gfCNCPoint4[22804] = {X 353.6578, Y 29.0247, Z -6.3333, A 0.000, B 0.000, C 0.000 }
gfCNCPoint4[22805] = {X 353.9952, Y 27.8508, Z -6.3333, A 0.000, B 0.000, C 0.000 }
gfCNCPoint4[22806] = {X 354.2226, Y 26.4400, Z -6.3333, A 0.000, B 0.000, C 0.000 }
gfCNCPoint4[22807] = {X 354.3146, Y 25.0140, Z -6.3333, A 0.000, B 0.000, C 0.000 }
gfCNCPoint4[22808] = {X 354.2704, Y 23.5857, Z -6.3333, A 0.000, B 0.000, C 0.000 }
gfCNCPoint4[22809] = {X 354.0904, Y 22.1681, Z -6.3333, A 0.000, B 0.000, C 0.000 }
gfCNCPoint4[22810] = {X 353.8255, Y 21.0252, Z -6.3333, A 0.000, B 0.000, C 0.000 }
gfCNCPoint4[22811] = {X 353.4123, Y 19.9272, Z -6.3333, A 0.000, B 0.000, C 0.000 }
gfCNCPoint4[22812] = {X 352.8578, Y 18.8933, Z -6.3333, A 0.000, B 0.000, C 0.000 }
gfCNCPoint4[22813] = {X 352.1719, Y 17.9415, Z -6.3333, A 0.000, B 0.000, C 0.000 }
gfCNCPoint4[22814] = {X 351.4219, Y 17.1684, Z -6.3333, A 0.000, B 0.000, C 0.000 }
gfCNCPoint4[22815] = {X 350.5492, Y 16.5370, Z -6.3333, A 0.000, B 0.000, C 0.000 }
gfCNCPoint4[22816] = {X 349.5803, Y 16.0665, Z -6.3333, A 0.000, B 0.000, C 0.000 }
gfCNCPoint4[22817] = {X 348.5445, Y 15.7710, Z -6.3333, A 0.000, B 0.000, C 0.000 }
gfCNCPoint4[22818] = {X 347.1584, Y 15.5990, Z -6.3333, A 0.000, B 0.000, C 0.000 }
gfCNCPoint4[22819] = {X 345.7616, Y 15.6142, Z -6.3333, A 0.000, B 0.000, C 0.000 }
gfCNCPoint4[22820] = {X 344.3795, Y 15.8164, Z -6.3333, A 0.000, B 0.000, C 0.000 }
gfCNCPoint4[22821] = {X 343.0370, Y 16.2019, Z -6.3333, A 0.000, B 0.000, C 0.000 }
gfCNCPoint4[22822] = {X 341.7582, Y 16.7639, Z -6.3333, A 0.000, B 0.000, C 0.000 }
gfCNCPoint4[22823] = {X 341.3707, Y 18.0084, Z -6.3333, A 0.000, B 0.000, C 0.000 }
gfCNCPoint4[22824] = {X 340.7675, Y 19.1639, Z -6.3333, A 0.000, B 0.000, C 0.000 }
gfCNCPoint4[22825] = {X 339.9680, Y 20.1933, Z -6.3333, A 0.000, B 0.000, C 0.000 }
gfCNCPoint4[22826] = {X 338.9976, Y 21.0636, Z -6.3333, A 0.000, B 0.000, C 0.000 }
gfCNCPoint4[22827] = {X 338.2497, Y 21.6140, Z -6.3333, A 0.000, B 0.000, C 0.000 }
gfCNCPoint4[22828] = {X 337.8538, Y 21.8795, Z -6.3333, A 0.000, B 0.000, C 0.000 }
gfCNCPoint4[22829] = {X 337.4413, Y 22.1185, Z -6.3333, A 0.000, B 0.000, C 0.000 }
gfCNCPoint4[22830] = {X 336.3239, Y 22.6023, Z -6.3333, A 0.000, B 0.000, C 0.000 }
gfCNCPoint4[22831] = {X 335.1415, Y 22.8932, Z -6.3333, A 0.000, B 0.000, C 0.000 }
gfCNCPoint4[22832] = {X 333.9271, Y 22.9829, Z -6.3333, A 0.000, B 0.000, C 0.000 }
gfCNCPoint4[22833] = {X 332.7148, Y 22.8690, Z -6.3333, A 0.000, B 0.000, C 0.000 }
gfCNCPoint4[22834] = {X 331.5384, Y 22.5546, Z -6.3333, A 0.000, B 0.000, C 0.000 }
gfCNCPoint4[22835] = {X 330.4309, Y 22.0485, Z -6.3333, A 0.000, B 0.000, C 0.000 }
gfCNCPoint4[22836] = {X 329.5143, Y 21.4374, Z -6.3333, A 0.000, B 0.000, C 0.000 }
gfCNCPoint4[22837] = {X 328.7005, Y 20.6949, Z -6.3333, A 0.000, B 0.000, C 0.000 }
gfCNCPoint4[22838] = {X 328.0080, Y 19.8382, Z -6.3333, A 0.000, B 0.000, C 0.000 }
gfCNCPoint4[22839] = {X 327.4528, Y 18.8869, Z -6.3333, A 0.000, B 0.000, C 0.000 }
gfCNCPoint4[22840] = {X 323.9321, Y 11.6443, Z -6.3333, A 0.000, B 0.000, C 0.000 }
gfCNCPoint4[22841] = {X 323.5337, Y 10.6421, Z -6.3333, A 0.000, B 0.000, C 0.000 }
gfCNCPoint4[22842] = {X 323.2878, Y 9.5921, Z -6.3333, A 0.000, B 0.000, C 0.000 }
gfCNCPoint4[22843] = {X 323.1997, Y 8.5173, Z -6.3333, A 0.000, B 0.000, C 0.000 }
gfCNCPoint4[22844] = {X 323.2713, Y 7.4413, Z -6.3333, A 0.000, B 0.000, C 0.000 }
gfCNCPoint4[22845] = {X 323.4720, Y 6.4884, Z -6.3333, A 0.000, B 0.000, C 0.000 }
gfCNCPoint4[22846] = {X 323.7980, Y 5.5708, Z -6.3333, A 0.000, B 0.000, C 0.000 }
gfCNCPoint4[22847] = {X 324.2436, Y 4.7049, Z -6.3333, A 0.000, B 0.000, C 0.000 }
gfCNCPoint4[22848] = {X 168.0206, Y 4.7049, Z -6.3333, A 0.000, B 0.000, C 0.000 }
gfCNCPoint4[22849] = {X 168.0206, Y 9.5049, Z -6.3333, A 0.000, B 0.000, C 0.000 }
gfCNCPoint4[22850] = {X 166.5360, Y 9.5049, Z -6.3333, A 0.000, B 0.000, C 0.000 }
gfCNCPoint4[22851] = {X 166.5855, Y 9.9931, Z -6.3333, A 0.000, B 0.000, C 0.000 }
gfCNCPoint4[22852] = {X 166.6021, Y 10.4835, Z -6.3333, A 0.000, B 0.000, C 0.000 }
gfCNCPoint4[22853] = {X 166.6021, Y 13.0969, Z -6.3333, A 0.000, B 0.000, C 0.000 }
gfCNCPoint4[22854] = {X 166.8569, Y 11.8209, Z -6.3333, A 0.000, B 0.000, C 0.000 }
gfCNCPoint4[22855] = {X 167.3349, Y 10.6107, Z -6.3333, A 0.000, B 0.000, C 0.000 }
gfCNCPoint4[22856] = {X 168.0206, Y 9.5049, Z -6.3333, A 0.000, B 0.000, C 0.000 }
gfCNCPoint4[22857] = {X 168.0206, Y 7.1049, Z -6.3333, A 0.000, B 0.000, C 0.000 }
gfCNCPoint4[22858] = {X 162.8434, Y 7.1049, Z -6.3333, A 0.000, B 0.000, C 0.000 }
gfCNCPoint4[22859] = {X 163.4702, Y 7.9130, Z -6.3333, A 0.000, B 0.000, C 0.000 }
gfCNCPoint4[22860] = {X 163.9149, Y 8.8340, Z -6.3333, A 0.000, B 0.000, C 0.000 }
gfCNCPoint4[22861] = {X 164.1578, Y 9.8275, Z -6.3333, A 0.000, B 0.000, C 0.000 }
gfCNCPoint4[22862] = {X 164.1910, Y 10.1548, Z -6.3333, A 0.000, B 0.000, C 0.000 }
gfCNCPoint4[22863] = {X 164.2021, Y 10.4835, Z -6.3333, A 0.000, B 0.000, C 0.000 }
gfCNCPoint4[22864] = {X 164.2021, Y 17.4615, Z -6.3333, A 0.000, B 0.000, C 0.000 }
gfCNCPoint4[22865] = {X 164.1140, Y 18.3847, Z -6.3333, A 0.000, B 0.000, C 0.000 }
gfCNCPoint4[22866] = {X 163.8528, Y 19.2745, Z -6.3333, A 0.000, B 0.000, C 0.000 }
gfCNCPoint4[22867] = {X 163.4280, Y 20.0989, Z -6.3333, A 0.000, B 0.000, C 0.000 }
gfCNCPoint4[22868] = {X 162.8550, Y 20.8280, Z -6.3333, A 0.000, B 0.000, C 0.000 }
gfCNCPoint4[22869] = {X 162.1544, Y 21.4355, Z -6.3333, A 0.000, B 0.000, C 0.000 }
gfCNCPoint4[22870] = {X 161.3515, Y 21.8996, Z -6.3333, A 0.000, B 0.000, C 0.000 }
gfCNCPoint4[22871] = {X 160.4753, Y 22.2033, Z -6.3333, A 0.000, B 0.000, C 0.000 }
gfCNCPoint4[22872] = {X 162.1767, Y 29.1994, Z -6.3333, A 0.000, B 0.000, C 0.000 }
gfCNCPoint4[22873] = {X 161.1138, Y 29.4079, Z -6.3333, A 0.000, B 0.000, C 0.000 }
gfCNCPoint4[22874] = {X 160.0364, Y 29.5204, Z -6.3333, A 0.000, B 0.000, C 0.000 }
gfCNCPoint4[22875] = {X 160.0359, Y 38.3363, Z -6.3333, A 0.000, B 0.000, C 0.000 }
gfCNCPoint4[22876] = {X 160.6841, Y 39.6935, Z -6.3333, A 0.000, B 0.000, C 0.000 }
gfCNCPoint4[22877] = {X 161.1590, Y 41.1206, Z -6.3333, A 0.000, B 0.000, C 0.000 }
gfCNCPoint4[22878] = {X 162.0525, Y 41.1205, Z -6.3333, A 0.000, B 0.000, C 0.000 }
gfCNCPoint4[22879] = {X 161.8701, Y 40.3466, Z -6.3333, A 0.000, B 0.000, C 0.000 }
gfCNCPoint4[22880] = {X 161.7176, Y 39.5664, Z -6.3333, A 0.000, B 0.000, C 0.000 }
gfCNCPoint4[22881] = {X 161.5943, Y 38.7924, Z -6.3333, A 0.000, B 0.000, C 0.000 }
gfCNCPoint4[22882] = {X 161.3800, Y 36.8680, Z -6.3333, A 0.000, B 0.000, C 0.000 }
gfCNCPoint4[22883] = {X 161.3313, Y 34.9322, Z -6.3333, A 0.000, B 0.000, C 0.000 }
gfCNCPoint4[22884] = {X 161.4486, Y 32.9994, Z -6.3333, A 0.000, B 0.000, C 0.000 }
gfCNCPoint4[22885] = {X 161.7311, Y 31.0838, Z -6.3333, A 0.000, B 0.000, C 0.000 }
gfCNCPoint4[22886] = {X 162.1767, Y 29.1994, Z -6.3333, A 0.000, B 0.000, C 0.000 }
gfCNCPoint4[22887] = {X 161.6096, Y 26.8674, Z -6.3333, A 0.000, B 0.000, C 0.000 }
gfCNCPoint4[22888] = {X 160.4740, Y 27.0728, Z -6.3333, A 0.000, B 0.000, C 0.000 }
gfCNCPoint4[22889] = {X 159.3220, Y 27.1415, Z -6.3333, A 0.000, B 0.000, C 0.000 }
gfCNCPoint4[22890] = {X 158.6595, Y 27.1415, Z -6.3333, A 0.000, B 0.000, C 0.000 }
gfCNCPoint4[22891] = {X 158.1473, Y 27.1261, Z -6.3333, A 0.000, B 0.000, C 0.000 }
gfCNCPoint4[22892] = {X 157.6365, Y 27.0837, Z -6.3333, A 0.000, B 0.000, C 0.000 }
gfCNCPoint4[22893] = {X 157.6359, Y 38.9959, Z -6.3333, A 0.000, B 0.000, C 0.000 }
gfCNCPoint4[22894] = {X 158.2197, Y 40.0483, Z -6.3333, A 0.000, B 0.000, C 0.000 }
gfCNCPoint4[22895] = {X 158.6689, Y 41.1648, Z -6.3333, A 0.000, B 0.000, C 0.000 }
gfCNCPoint4[22896] = {X 158.9765, Y 42.3283, Z -6.3333, A 0.000, B 0.000, C 0.000 }
gfCNCPoint4[22897] = {X 159.1377, Y 43.5209, Z -6.3333, A 0.000, B 0.000, C 0.000 }
gfCNCPoint4[22898] = {X 165.4263, Y 43.5200, Z -6.3333, A 0.000, B 0.000, C 0.000 }
gfCNCPoint4[22899] = {X 164.8372, Y 42.0454, Z -6.3333, A 0.000, B 0.000, C 0.000 }
gfCNCPoint4[22900] = {X 164.3775, Y 40.5256, Z -6.3333, A 0.000, B 0.000, C 0.000 }
gfCNCPoint4[22901] = {X 164.2182, Y 39.8499, Z -6.3333, A 0.000, B 0.000, C 0.000 }
gfCNCPoint4[22902] = {X 164.0845, Y 39.1688, Z -6.3333, A 0.000, B 0.000, C 0.000 }
gfCNCPoint4[22903] = {X 163.9653, Y 38.4202, Z -6.3333, A 0.000, B 0.000, C 0.000 }
gfCNCPoint4[22904] = {X 163.7495, Y 36.2693, Z -6.3333, A 0.000, B 0.000, C 0.000 }
gfCNCPoint4[22905] = {X 163.7649, Y 34.1077, Z -6.3333, A 0.000, B 0.000, C 0.000 }
gfCNCPoint4[22906] = {X 164.0116, Y 31.9602, Z -6.3333, A 0.000, B 0.000, C 0.000 }
gfCNCPoint4[22907] = {X 164.4865, Y 29.8513, Z -6.3333, A 0.000, B 0.000, C 0.000 }
gfCNCPoint4[22908] = {X 164.8367, Y 28.7352, Z -6.3333, A 0.000, B 0.000, C 0.000 }
gfCNCPoint4[22909] = {X 165.2511, Y 27.6412, Z -6.3333, A 0.000, B 0.000, C 0.000 }
gfCNCPoint4[22910] = {X 165.8680, Y 26.3084, Z -6.3333, A 0.000, B 0.000, C 0.000 }
gfCNCPoint4[22911] = {X 166.6029, Y 25.0369, Z -6.3333, A 0.000, B 0.000, C 0.000 }
gfCNCPoint4[22912] = {X 167.4499, Y 23.8371, Z -6.3333, A 0.000, B 0.000, C 0.000 }
gfCNCPoint4[22913] = {X 167.1640, Y 23.1367, Z -6.3333, A 0.000, B 0.000, C 0.000 }
gfCNCPoint4[22914] = {X 166.2875, Y 24.1835, Z -6.3333, A 0.000, B 0.000, C 0.000 }
gfCNCPoint4[22915] = {X 165.2726, Y 25.0966, Z -6.3333, A 0.000, B 0.000, C 0.000 }
gfCNCPoint4[22916] = {X 164.1393, Y 25.8578, Z -6.3333, A 0.000, B 0.000, C 0.000 }
gfCNCPoint4[22917] = {X 162.9101, Y 26.4520, Z -6.3333, A 0.000, B 0.000, C 0.000 }
gfCNCPoint4[22918] = {X 161.6096, Y 26.8674, Z -6.3333, A 0.000, B 0.000, C 0.000 }
gfCNCPoint4[22919] = {X 161.0424, Y 24.5353, Z -6.3333, A 0.000, B 0.000, C 0.000 }
gfCNCPoint4[22920] = {X 160.1884, Y 24.6898, Z -6.3333, A 0.000, B 0.000, C 0.000 }
gfCNCPoint4[22921] = {X 159.3220, Y 24.7415, Z -6.3333, A 0.000, B 0.000, C 0.000 }
gfCNCPoint4[22922] = {X 158.6684, Y 24.7415, Z -6.3333, A 0.000, B 0.000, C 0.000 }
gfCNCPoint4[22923] = {X 158.2827, Y 24.7299, Z -6.3333, A 0.000, B 0.000, C 0.000 }
gfCNCPoint4[22924] = {X 157.8982, Y 24.6980, Z -6.3333, A 0.000, B 0.000, C 0.000 }
gfCNCPoint4[22925] = {X 156.9782, Y 24.5371, Z -6.3333, A 0.000, B 0.000, C 0.000 }
gfCNCPoint4[22926] = {X 156.0862, Y 24.2602, Z -6.3333, A 0.000, B 0.000, C 0.000 }
gfCNCPoint4[22927] = {X 155.2367, Y 23.8718, Z -6.3333, A 0.000, B 0.000, C 0.000 }
gfCNCPoint4[22928] = {X 155.2358, Y 39.7518, Z -6.3333, A 0.000, B 0.000, C 0.000 }
gfCNCPoint4[22929] = {X 155.8266, Y 40.6435, Z -6.3333, A 0.000, B 0.000, C 0.000 }
gfCNCPoint4[22930] = {X 156.2808, Y 41.6118, Z -6.3333, A 0.000, B 0.000, C 0.000 }
gfCNCPoint4[22931] = {X 156.5888, Y 42.6361, Z -6.3333, A 0.000, B 0.000, C 0.000 }
gfCNCPoint4[22932] = {X 156.7440, Y 43.6944, Z -6.3333, A 0.000, B 0.000, C 0.000 }
gfCNCPoint4[22933] = {X 156.7580, Y 43.9481, Z -6.3333, A 0.000, B 0.000, C 0.000 }
gfCNCPoint4[22934] = {X 156.7631, Y 44.2022, Z -6.3333, A 0.000, B 0.000, C 0.000 }
gfCNCPoint4[22935] = {X 156.7629, Y 45.0588, Z -6.3333, A 0.000, B 0.000, C 0.000 }
gfCNCPoint4[22936] = {X 156.7352, Y 45.6370, Z -6.3333, A 0.000, B 0.000, C 0.000 }
gfCNCPoint4[22937] = {X 156.6616, Y 46.2112, Z -6.3333, A 0.000, B 0.000, C 0.000 }
gfCNCPoint4[22938] = {X 157.9054, Y 46.0005, Z -6.3333, A 0.000, B 0.000, C 0.000 }
gfCNCPoint4[22939] = {X 159.1643, Y 45.9207, Z -6.3333, A 0.000, B 0.000, C 0.000 }
gfCNCPoint4[22940] = {X 159.2311, Y 45.9202, Z -6.3333, A 0.000, B 0.000, C 0.000 }
gfCNCPoint4[22941] = {X 159.2980, Y 45.9200, Z -6.3333, A 0.000, B 0.000, C 0.000 }
gfCNCPoint4[22942] = {X 169.6793, Y 45.9200, Z -6.3333, A 0.000, B 0.000, C 0.000 }
gfCNCPoint4[22943] = {X 168.8981, Y 44.8498, Z -6.3333, A 0.000, B 0.000, C 0.000 }
gfCNCPoint4[22944] = {X 168.2083, Y 43.7186, Z -6.3333, A 0.000, B 0.000, C 0.000 }
gfCNCPoint4[22945] = {X 167.6145, Y 42.5342, Z -6.3333, A 0.000, B 0.000, C 0.000 }
gfCNCPoint4[22946] = {X 167.1237, Y 41.3128, Z -6.3333, A 0.000, B 0.000, C 0.000 }
gfCNCPoint4[22947] = {X 166.7350, Y 40.0551, Z -6.3333, A 0.000, B 0.000, C 0.000 }
gfCNCPoint4[22948] = {X 166.4512, Y 38.7697, Z -6.3333, A 0.000, B 0.000, C 0.000 }
gfCNCPoint4[22949] = {X 166.3363, Y 38.0482, Z -6.3333, A 0.000, B 0.000, C 0.000 }
gfCNCPoint4[22950] = {X 166.1452, Y 36.1222, Z -6.3333, A 0.000, B 0.000, C 0.000 }
gfCNCPoint4[22951] = {X 166.1647, Y 34.1868, Z -6.3333, A 0.000, B 0.000, C 0.000 }
gfCNCPoint4[22952] = {X 166.3944, Y 32.2650, Z -6.3333, A 0.000, B 0.000, C 0.000 }
gfCNCPoint4[22953] = {X 166.8316, Y 30.3795, Z -6.3333, A 0.000, B 0.000, C 0.000 }
gfCNCPoint4[22954] = {X 167.4712, Y 28.5528, Z -6.3333, A 0.000, B 0.000, C 0.000 }
gfCNCPoint4[22955] = {X 168.2320, Y 26.9825, Z -6.3333, A 0.000, B 0.000, C 0.000 }
gfCNCPoint4[22956] = {X 169.1846, Y 25.5206, Z -6.3333, A 0.000, B 0.000, C 0.000 }
gfCNCPoint4[22957] = {X 170.3139, Y 24.1904, Z -6.3333, A 0.000, B 0.000, C 0.000 }
gfCNCPoint4[22958] = {X 169.9864, Y 23.6220, Z -6.3333, A 0.000, B 0.000, C 0.000 }
gfCNCPoint4[22959] = {X 169.7113, Y 23.0264, Z -6.3333, A 0.000, B 0.000, C 0.000 }
gfCNCPoint4[22960] = {X 167.1001, Y 16.6309, Z -6.3333, A 0.000, B 0.000, C 0.000 }
gfCNCPoint4[22961] = {X 166.7820, Y 15.6636, Z -6.3333, A 0.000, B 0.000, C 0.000 }
gfCNCPoint4[22962] = {X 166.6021, Y 14.6613, Z -6.3333, A 0.000, B 0.000, C 0.000 }
gfCNCPoint4[22963] = {X 166.6021, Y 17.4615, Z -6.3333, A 0.000, B 0.000, C 0.000 }
gfCNCPoint4[22964] = {X 166.5130, Y 18.5970, Z -6.3333, A 0.000, B 0.000, C 0.000 }
gfCNCPoint4[22965] = {X 166.2479, Y 19.7047, Z -6.3333, A 0.000, B 0.000, C 0.000 }
gfCNCPoint4[22966] = {X 165.8132, Y 20.7575, Z -6.3333, A 0.000, B 0.000, C 0.000 }
gfCNCPoint4[22967] = {X 165.2197, Y 21.7296, Z -6.3333, A 0.000, B 0.000, C 0.000 }
gfCNCPoint4[22968] = {X 164.3790, Y 22.6986, Z -6.3333, A 0.000, B 0.000, C 0.000 }
gfCNCPoint4[22969] = {X 163.3812, Y 23.5049, Z -6.3333, A 0.000, B 0.000, C 0.000 }
gfCNCPoint4[22970] = {X 162.2574, Y 24.1236, Z -6.3333, A 0.000, B 0.000, C 0.000 }
gfCNCPoint4[22971] = {X 161.0424, Y 24.5353, Z -6.3333, A 0.000, B 0.000, C 0.000 }
gfCNCPoint4[22972] = {X 160.4753, Y 22.2033, Z -6.3333, A 0.000, B 0.000, C 0.000 }
gfCNCPoint4[22973] = {X 159.9028, Y 22.3069, Z -6.3333, A 0.000, B 0.000, C 0.000 }
gfCNCPoint4[22974] = {X 159.3220, Y 22.3415, Z -6.3333, A 0.000, B 0.000, C 0.000 }
gfCNCPoint4[22975] = {X 158.6772, Y 22.3415, Z -6.3333, A 0.000, B 0.000, C 0.000 }
gfCNCPoint4[22976] = {X 157.8803, Y 22.2735, Z -6.3333, A 0.000, B 0.000, C 0.000 }
gfCNCPoint4[22977] = {X 157.1051, Y 22.0770, Z -6.3333, A 0.000, B 0.000, C 0.000 }
gfCNCPoint4[22978] = {X 156.3720, Y 21.7573, Z -6.3333, A 0.000, B 0.000, C 0.000 }
gfCNCPoint4[22979] = {X 155.5228, Y 21.1795, Z -6.3333, A 0.000, B 0.000, C 0.000 }
gfCNCPoint4[22980] = {X 154.8124, Y 20.4377, Z -6.3333, A 0.000, B 0.000, C 0.000 }
gfCNCPoint4[22981] = {X 152.8369, Y 20.4384, Z -6.3333, A 0.000, B 0.000, C 0.000 }
gfCNCPoint4[22982] = {X 152.8358, Y 40.6543, Z -6.3333, A 0.000, B 0.000, C 0.000 }
gfCNCPoint4[22983] = {X 153.1748, Y 41.0209, Z -6.3333, A 0.000, B 0.000, C 0.000 }
gfCNCPoint4[22984] = {X 153.6800, Y 41.7251, Z -6.3333, A 0.000, B 0.000, C 0.000 }
gfCNCPoint4[22985] = {X 154.0535, Y 42.5072, Z -6.3333, A 0.000, B 0.000, C 0.000 }
gfCNCPoint4[22986] = {X 154.2836, Y 43.3429, Z -6.3333, A 0.000, B 0.000, C 0.000 }
gfCNCPoint4[22987] = {X 154.3631, Y 44.2060, Z -6.3333, A 0.000, B 0.000, C 0.000 }
gfCNCPoint4[22988] = {X 154.3629, Y 45.0469, Z -6.3333, A 0.000, B 0.000, C 0.000 }
gfCNCPoint4[22989] = {X 154.3440, Y 45.4308, Z -6.3333, A 0.000, B 0.000, C 0.000 }
gfCNCPoint4[22990] = {X 154.2951, Y 45.8119, Z -6.3333, A 0.000, B 0.000, C 0.000 }
gfCNCPoint4[22991] = {X 154.0370, Y 46.7541, Z -6.3333, A 0.000, B 0.000, C 0.000 }
gfCNCPoint4[22992] = {X 153.5963, Y 47.6260, Z -6.3333, A 0.000, B 0.000, C 0.000 }
gfCNCPoint4[22993] = {X 152.9909, Y 48.3926, Z -6.3333, A 0.000, B 0.000, C 0.000 }
gfCNCPoint4[22994] = {X 152.2448, Y 49.0233, Z -6.3333, A 0.000, B 0.000, C 0.000 }
gfCNCPoint4[22995] = {X 151.3881, Y 49.4928, Z -6.3333, A 0.000, B 0.000, C 0.000 }
gfCNCPoint4[22996] = {X 150.4551, Y 49.7822, Z -6.3333, A 0.000, B 0.000, C 0.000 }
gfCNCPoint4[22997] = {X 149.4831, Y 49.8800, Z -6.3333, A 0.000, B 0.000, C 0.000 }
gfCNCPoint4[22998] = {X 143.0396, Y 49.8800, Z -6.3333, A 0.000, B 0.000, C 0.000 }
gfCNCPoint4[22999] = {X 142.0923, Y 49.7872, Z -6.3333, A 0.000, B 0.000, C 0.000 }
gfCNCPoint4[23000] = {X 141.1811, Y 49.5122, Z -6.3333, A 0.000, B 0.000, C 0.000 }
gfCNCPoint4[23001] = {X 140.3405, Y 49.0656, Z -6.3333, A 0.000, B 0.000, C 0.000 }
gfCNCPoint4[23002] = {X 139.6026, Y 48.4643, Z -6.3333, A 0.000, B 0.000, C 0.000 }
gfCNCPoint4[23003] = {X 138.9955, Y 47.7312, Z -6.3333, A 0.000, B 0.000, C 0.000 }
gfCNCPoint4[23004] = {X 138.5423, Y 46.8942, Z -6.3333, A 0.000, B 0.000, C 0.000 }
gfCNCPoint4[23005] = {X 138.2601, Y 45.9852, Z -6.3333, A 0.000, B 0.000, C 0.000 }
gfCNCPoint4[23006] = {X 138.1598, Y 45.0386, Z -6.3333, A 0.000, B 0.000, C 0.000 }
gfCNCPoint4[23007] = {X 138.1601, Y 44.1416, Z -6.3333, A 0.000, B 0.000, C 0.000 }
gfCNCPoint4[23008] = {X 138.2148, Y 43.4769, Z -6.3333, A 0.000, B 0.000, C 0.000 }
gfCNCPoint4[23009] = {X 138.3597, Y 42.8258, Z -6.3333, A 0.000, B 0.000, C 0.000 }
gfCNCPoint4[23010] = {X 129.1532, Y 40.1052, Z -6.3333, A 0.000, B 0.000, C 0.000 }
gfCNCPoint4[23011] = {X 129.5665, Y 38.9035, Z -6.3333, A 0.000, B 0.000, C 0.000 }
gfCNCPoint4[23012] = {X 130.0836, Y 37.7426, Z -6.3333, A 0.000, B 0.000, C 0.000 }
gfCNCPoint4[23013] = {X 130.0836, Y 31.6021, Z -6.3333, A 0.000, B 0.000, C 0.000 }
gfCNCPoint4[23014] = {X 129.2064, Y 31.3798, Z -6.3333, A 0.000, B 0.000, C 0.000 }
gfCNCPoint4[23015] = {X 128.3449, Y 31.1031, Z -6.3333, A 0.000, B 0.000, C 0.000 }
gfCNCPoint4[23016] = {X 128.3447, Y 38.3302, Z -6.3333, A 0.000, B 0.000, C 0.000 }
gfCNCPoint4[23017] = {X 128.7849, Y 39.2014, Z -6.3333, A 0.000, B 0.000, C 0.000 }
gfCNCPoint4[23018] = {X 129.1532, Y 40.1052, Z -6.3333, A 0.000, B 0.000, C 0.000 }
gfCNCPoint4[23019] = {X 131.4548, Y 40.7854, Z -6.3333, A 0.000, B 0.000, C 0.000 }
gfCNCPoint4[23020] = {X 131.9017, Y 39.5320, Z -6.3333, A 0.000, B 0.000, C 0.000 }
gfCNCPoint4[23021] = {X 132.4836, Y 38.3354, Z -6.3333, A 0.000, B 0.000, C 0.000 }
gfCNCPoint4[23022] = {X 132.4836, Y 29.5202, Z -6.3333, A 0.000, B 0.000, C 0.000 }
gfCNCPoint4[23023] = {X 131.3526, Y 29.3993, Z -6.3333, A 0.000, B 0.000, C 0.000 }
gfCNCPoint4[23024] = {X 130.2380, Y 29.1726, Z -6.3333, A 0.000, B 0.000, C 0.000 }
gfCNCPoint4[23025] = {X 129.1497, Y 28.8421, Z -6.3333, A 0.000, B 0.000, C 0.000 }
gfCNCPoint4[23026] = {X 128.0253, Y 28.3768, Z -6.3333, A 0.000, B 0.000, C 0.000 }
gfCNCPoint4[23027] = {X 126.9534, Y 27.8007, Z -6.3333, A 0.000, B 0.000, C 0.000 }
gfCNCPoint4[23028] = {X 125.9449, Y 27.1197, Z -6.3333, A 0.000, B 0.000, C 0.000 }
gfCNCPoint4[23029] = {X 125.9447, Y 38.9907, Z -6.3333, A 0.000, B 0.000, C 0.000 }
gfCNCPoint4[23030] = {X 126.4741, Y 39.9291, Z -6.3333, A 0.000, B 0.000, C 0.000 }
gfCNCPoint4[23031] = {X 126.8960, Y 40.9205, Z -6.3333, A 0.000, B 0.000, C 0.000 }
gfCNCPoint4[23032] = {X 127.2098, Y 41.9730, Z -6.3333, A 0.000, B 0.000, C 0.000 }
gfCNCPoint4[23033] = {X 127.4025, Y 43.0542, Z -6.3333, A 0.000, B 0.000, C 0.000 }
gfCNCPoint4[23034] = {X 127.4714, Y 44.1502, Z -6.3333, A 0.000, B 0.000, C 0.000 }
gfCNCPoint4[23035] = {X 127.4716, Y 45.0000, Z -6.3333, A 0.000, B 0.000, C 0.000 }
gfCNCPoint4[23036] = {X 127.4070, Y 46.1159, Z -6.3333, A 0.000, B 0.000, C 0.000 }
gfCNCPoint4[23037] = {X 127.2143, Y 47.2168, Z -6.3333, A 0.000, B 0.000, C 0.000 }
gfCNCPoint4[23038] = {X 126.8960, Y 48.2883, Z -6.3333, A 0.000, B 0.000, C 0.000 }
gfCNCPoint4[23039] = {X 126.2883, Y 49.6376, Z -6.3333, A 0.000, B 0.000, C 0.000 }
gfCNCPoint4[23040] = {X 125.4821, Y 50.8786, Z -6.3333, A 0.000, B 0.000, C 0.000 }
gfCNCPoint4[23041] = {X 124.4962, Y 51.9821, Z -6.3333, A 0.000, B 0.000, C 0.000 }
gfCNCPoint4[23042] = {X 123.3536, Y 52.9225, Z -6.3333, A 0.000, B 0.000, C 0.000 }
gfCNCPoint4[23043] = {X 122.0810, Y 53.6778, Z -6.3333, A 0.000, B 0.000, C 0.000 }
gfCNCPoint4[23044] = {X 120.7081, Y 54.2302, Z -6.3333, A 0.000, B 0.000, C 0.000 }
gfCNCPoint4[23045] = {X 119.2671, Y 54.5669, Z -6.3333, A 0.000, B 0.000, C 0.000 }
gfCNCPoint4[23046] = {X 117.7916, Y 54.6800, Z -6.3333, A 0.000, B 0.000, C 0.000 }
gfCNCPoint4[23047] = {X 111.9185, Y 54.6800, Z -6.3333, A 0.000, B 0.000, C 0.000 }
gfCNCPoint4[23048] = {X 111.7456, Y 54.6785, Z -6.3333, A 0.000, B 0.000, C 0.000 }
gfCNCPoint4[23049] = {X 111.5728, Y 54.6738, Z -6.3333, A 0.000, B 0.000, C 0.000 }
gfCNCPoint4[23050] = {X 111.0585, Y 69.0646, Z -6.3333, A 0.000, B 0.000, C 0.000 }
gfCNCPoint4[23051] = {X 109.0296, Y 68.9061, Z -6.3333, A 0.000, B 0.000, C 0.000 }
gfCNCPoint4[23052] = {X 107.0213, Y 68.5768, Z -6.3333, A 0.000, B 0.000, C 0.000 }
gfCNCPoint4[23053] = {X 105.0765, Y 68.8983, Z -6.3333, A 0.000, B 0.000, C 0.000 }
gfCNCPoint4[23054] = {X 103.1119, Y 69.0597, Z -6.3333, A 0.000, B 0.000, C 0.000 }
gfCNCPoint4[23055] = {X 101.1407, Y 69.0599, Z -6.3333, A 0.000, B 0.000, C 0.000 }
gfCNCPoint4[23056] = {X 99.1761, Y 68.8989, Z -6.3333, A 0.000, B 0.000, C 0.000 }
gfCNCPoint4[23057] = {X 97.2313, Y 68.5777, Z -6.3333, A 0.000, B 0.000, C 0.000 }
gfCNCPoint4[23058] = {X 95.6131, Y 68.8563, Z -6.3333, A 0.000, B 0.000, C 0.000 }
gfCNCPoint4[23059] = {X 93.9796, Y 69.0240, Z -6.3333, A 0.000, B 0.000, C 0.000 }
gfCNCPoint4[23060] = {X 92.3385, Y 69.0800, Z -6.3333, A 0.000, B 0.000, C 0.000 }
gfCNCPoint4[23061] = {X 86.6884, Y 69.0800, Z -6.3333, A 0.000, B 0.000, C 0.000 }
gfCNCPoint4[23062] = {X 84.7316, Y 70.2669, Z -6.3333, A 0.000, B 0.000, C 0.000 }
gfCNCPoint4[23063] = {X 82.6869, Y 71.2951, Z -6.3333, A 0.000, B 0.000, C 0.000 }
gfCNCPoint4[23064] = {X 107.2714, Y 71.2951, Z -6.3333, A 0.000, B 0.000, C 0.000 }
gfCNCPoint4[23065] = {X 109.1257, Y 70.1133, Z -6.3333, A 0.000, B 0.000, C 0.000 }
gfCNCPoint4[23066] = {X 111.0585, Y 69.0646, Z -6.3333, A 0.000, B 0.000, C 0.000 }
gfCNCPoint4[23067] = {X 111.1442, Y 66.6662, Z -6.3333, A 0.000, B 0.000, C 0.000 }
gfCNCPoint4[23068] = {X 109.0696, Y 66.4920, Z -6.3333, A 0.000, B 0.000, C 0.000 }
gfCNCPoint4[23069] = {X 107.0213, Y 66.1197, Z -6.3333, A 0.000, B 0.000, C 0.000 }
gfCNCPoint4[23070] = {X 105.0796, Y 66.4776, Z -6.3333, A 0.000, B 0.000, C 0.000 }
gfCNCPoint4[23071] = {X 103.1135, Y 66.6574, Z -6.3333, A 0.000, B 0.000, C 0.000 }
gfCNCPoint4[23072] = {X 101.1392, Y 66.6576, Z -6.3333, A 0.000, B 0.000, C 0.000 }
gfCNCPoint4[23073] = {X 99.1730, Y 66.4782, Z -6.3333, A 0.000, B 0.000, C 0.000 }
gfCNCPoint4[23074] = {X 97.2313, Y 66.1207, Z -6.3333, A 0.000, B 0.000, C 0.000 }
gfCNCPoint4[23075] = {X 95.6161, Y 66.4308, Z -6.3333, A 0.000, B 0.000, C 0.000 }
gfCNCPoint4[23076] = {X 93.9821, Y 66.6176, Z -6.3333, A 0.000, B 0.000, C 0.000 }
gfCNCPoint4[23077] = {X 92.3385, Y 66.6800, Z -6.3333, A 0.000, B 0.000, C 0.000 }
gfCNCPoint4[23078] = {X 85.9487, Y 66.6800, Z -6.3333, A 0.000, B 0.000, C 0.000 }
gfCNCPoint4[23079] = {X 83.8779, Y 67.9936, Z -6.3333, A 0.000, B 0.000, C 0.000 }
gfCNCPoint4[23080] = {X 81.6945, Y 69.1099, Z -6.3333, A 0.000, B 0.000, C 0.000 }
gfCNCPoint4[23081] = {X 79.6015, Y 69.9548, Z -6.3333, A 0.000, B 0.000, C 0.000 }
gfCNCPoint4[23082] = {X 77.4442, Y 70.6184, Z -6.3333, A 0.000, B 0.000, C 0.000 }
gfCNCPoint4[23083] = {X 75.2382, Y 71.0959, Z -6.3333, A 0.000, B 0.000, C 0.000 }
gfCNCPoint4[23084] = {X 72.9995, Y 71.3838, Z -6.3333, A 0.000, B 0.000, C 0.000 }
gfCNCPoint4[23085] = {X 70.7445, Y 71.4800, Z -6.3333, A 0.000, B 0.000, C 0.000 }
gfCNCPoint4[23086] = {X 64.1851, Y 71.4800, Z -6.3333, A 0.000, B 0.000, C 0.000 }
gfCNCPoint4[23087] = {X 62.0752, Y 71.3958, Z -6.3333, A 0.000, B 0.000, C 0.000 }
gfCNCPoint4[23088] = {X 59.9787, Y 71.1438, Z -6.3333, A 0.000, B 0.000, C 0.000 }
gfCNCPoint4[23089] = {X 57.9089, Y 70.7255, Z -6.3333, A 0.000, B 0.000, C 0.000 }
gfCNCPoint4[23090] = {X 55.8790, Y 70.1436, Z -6.3333, A 0.000, B 0.000, C 0.000 }
gfCNCPoint4[23091] = {X 53.8492, Y 70.7255, Z -6.3333, A 0.000, B 0.000, C 0.000 }
gfCNCPoint4[23092] = {X 51.7794, Y 71.1438, Z -6.3333, A 0.000, B 0.000, C 0.000 }
gfCNCPoint4[23093] = {X 49.6829, Y 71.3958, Z -6.3333, A 0.000, B 0.000, C 0.000 }
gfCNCPoint4[23094] = {X 47.5729, Y 71.4800, Z -6.3333, A 0.000, B 0.000, C 0.000 }
gfCNCPoint4[23095] = {X 40.6393, Y 71.4800, Z -6.3333, A 0.000, B 0.000, C 0.000 }
gfCNCPoint4[23096] = {X 38.8056, Y 71.4164, Z -6.3333, A 0.000, B 0.000, C 0.000 }
gfCNCPoint4[23097] = {X 36.9807, Y 71.2260, Z -6.3333, A 0.000, B 0.000, C 0.000 }
gfCNCPoint4[23098] = {X 34.3981, Y 72.0359, Z -6.3333, A 0.000, B 0.000, C 0.000 }
gfCNCPoint4[23099] = {X 31.7544, Y 72.6161, Z -6.3333, A 0.000, B 0.000, C 0.000 }
gfCNCPoint4[23100] = {X 30.3306, Y 73.1752, Z -6.3333, A 0.000, B 0.000, C 0.000 }
gfCNCPoint4[23101] = {X 28.8922, Y 73.6951, Z -6.3333, A 0.000, B 0.000, C 0.000 }
gfCNCPoint4[23102] = {X 108.0336, Y 73.6951, Z -6.3333, A 0.000, B 0.000, C 0.000 }
gfCNCPoint4[23103] = {X 110.0294, Y 72.3691, Z -6.3333, A 0.000, B 0.000, C 0.000 }
gfCNCPoint4[23104] = {X 112.1282, Y 71.2131, Z -6.3333, A 0.000, B 0.000, C 0.000 }
gfCNCPoint4[23105] = {X 113.1260, Y 70.7398, Z -6.3333, A 0.000, B 0.000, C 0.000 }
gfCNCPoint4[23106] = {X 114.1413, Y 70.3051, Z -6.3333, A 0.000, B 0.000, C 0.000 }
gfCNCPoint4[23107] = {X 117.4424, Y 66.6800, Z -6.3333, A 0.000, B 0.000, C 0.000 }
gfCNCPoint4[23108] = {X 111.9185, Y 66.6800, Z -6.3333, A 0.000, B 0.000, C 0.000 }
gfCNCPoint4[23109] = {X 111.5313, Y 66.6765, Z -6.3333, A 0.000, B 0.000, C 0.000 }
gfCNCPoint4[23110] = {X 111.1442, Y 66.6662, Z -6.3333, A 0.000, B 0.000, C 0.000 }
gfCNCPoint4[23111] = {X 111.2299, Y 64.2677, Z -6.3333, A 0.000, B 0.000, C 0.000 }
gfCNCPoint4[23112] = {X 109.1084, Y 64.0741, Z -6.3333, A 0.000, B 0.000, C 0.000 }
gfCNCPoint4[23113] = {X 107.0213, Y 63.6477, Z -6.3333, A 0.000, B 0.000, C 0.000 }
gfCNCPoint4[23114] = {X 105.0841, Y 64.0514, Z -6.3333, A 0.000, B 0.000, C 0.000 }
gfCNCPoint4[23115] = {X 103.1158, Y 64.2545, Z -6.3333, A 0.000, B 0.000, C 0.000 }
gfCNCPoint4[23116] = {X 101.1370, Y 64.2547, Z -6.3333, A 0.000, B 0.000, C 0.000 }
gfCNCPoint4[23117] = {X 99.1686, Y 64.0521, Z -6.3333, A 0.000, B 0.000, C 0.000 }
gfCNCPoint4[23118] = {X 97.2313, Y 63.6488, Z -6.3333, A 0.000, B 0.000, C 0.000 }
gfCNCPoint4[23119] = {X 95.6204, Y 63.9986, Z -6.3333, A 0.000, B 0.000, C 0.000 }
gfCNCPoint4[23120] = {X 93.9855, Y 64.2095, Z -6.3333, A 0.000, B 0.000, C 0.000 }
gfCNCPoint4[23121] = {X 92.3385, Y 64.2800, Z -6.3333, A 0.000, B 0.000, C 0.000 }
gfCNCPoint4[23122] = {X 85.8951, Y 64.2800, Z -6.3333, A 0.000, B 0.000, C 0.000 }
gfCNCPoint4[23123] = {X 85.5417, Y 64.2768, Z -6.3333, A 0.000, B 0.000, C 0.000 }
gfCNCPoint4[23124] = {X 85.1884, Y 64.2670, Z -6.3333, A 0.000, B 0.000, C 0.000 }
gfCNCPoint4[23125] = {X 83.3593, Y 65.5113, Z -6.3333, A 0.000, B 0.000, C 0.000 }
gfCNCPoint4[23126] = {X 81.4238, Y 66.5824, Z -6.3333, A 0.000, B 0.000, C 0.000 }
gfCNCPoint4[23127] = {X 79.3981, Y 67.4713, Z -6.3333, A 0.000, B 0.000, C 0.000 }
gfCNCPoint4[23128] = {X 77.2994, Y 68.1706, Z -6.3333, A 0.000, B 0.000, C 0.000 }
gfCNCPoint4[23129] = {X 75.1454, Y 68.6744, Z -6.3333, A 0.000, B 0.000, C 0.000 }
gfCNCPoint4[23130] = {X 72.9543, Y 68.9784, Z -6.3333, A 0.000, B 0.000, C 0.000 }
gfCNCPoint4[23131] = {X 70.7445, Y 69.0800, Z -6.3333, A 0.000, B 0.000, C 0.000 }
gfCNCPoint4[23132] = {X 64.1851, Y 69.0800, Z -6.3333, A 0.000, B 0.000, C 0.000 }
gfCNCPoint4[23133] = {X 62.0678, Y 68.9867, Z -6.3333, A 0.000, B 0.000, C 0.000 }
gfCNCPoint4[23134] = {X 59.9669, Y 68.7076, Z -6.3333, A 0.000, B 0.000, C 0.000 }
gfCNCPoint4[23135] = {X 57.8986, Y 68.2449, Z -6.3333, A 0.000, B 0.000, C 0.000 }
gfCNCPoint4[23136] = {X 55.8790, Y 67.6021, Z -6.3333, A 0.000, B 0.000, C 0.000 }
gfCNCPoint4[23137] = {X 53.8595, Y 68.2449, Z -6.3333, A 0.000, B 0.000, C 0.000 }
gfCNCPoint4[23138] = {X 51.7912, Y 68.7076, Z -6.3333, A 0.000, B 0.000, C 0.000 }
gfCNCPoint4[23139] = {X 49.6903, Y 68.9867, Z -6.3333, A 0.000, B 0.000, C 0.000 }
gfCNCPoint4[23140] = {X 47.5729, Y 69.0800, Z -6.3333, A 0.000, B 0.000, C 0.000 }
gfCNCPoint4[23141] = {X 40.6393, Y 69.0800, Z -6.3333, A 0.000, B 0.000, C 0.000 }
gfCNCPoint4[23142] = {X 38.6751, Y 68.9998, Z -6.3333, A 0.000, B 0.000, C 0.000 }
gfCNCPoint4[23143] = {X 36.7239, Y 68.7596, Z -6.3333, A 0.000, B 0.000, C 0.000 }
gfCNCPoint4[23144] = {X 34.8824, Y 69.3998, Z -6.3333, A 0.000, B 0.000, C 0.000 }
gfCNCPoint4[23145] = {X 33.0012, Y 69.9123, Z -6.3333, A 0.000, B 0.000, C 0.000 }
gfCNCPoint4[23146] = {X 31.0893, Y 70.2945, Z -6.3333, A 0.000, B 0.000, C 0.000 }
gfCNCPoint4[23147] = {X 29.6068, Y 70.8830, Z -6.3333, A 0.000, B 0.000, C 0.000 }
gfCNCPoint4[23148] = {X 28.1074, Y 71.4270, Z -6.3333, A 0.000, B 0.000, C 0.000 }
gfCNCPoint4[23149] = {X 27.6130, Y 71.5954, Z -6.3333, A 0.000, B 0.000, C 0.000 }
gfCNCPoint4[23150] = {X 27.1170, Y 71.7589, Z -6.3333, A 0.000, B 0.000, C 0.000 }
gfCNCPoint4[23151] = {X 25.5185, Y 72.2527, Z -6.3333, A 0.000, B 0.000, C 0.000 }
gfCNCPoint4[23152] = {X 23.9034, Y 72.6890, Z -6.3333, A 0.000, B 0.000, C 0.000 }
gfCNCPoint4[23153] = {X 23.9034, Y 76.0951, Z -6.3333, A 0.000, B 0.000, C 0.000 }
gfCNCPoint4[23154] = {X 108.8317, Y 76.0951, Z -6.3333, A 0.000, B 0.000, C 0.000 }
gfCNCPoint4[23155] = {X 110.4015, Y 74.9736, Z -6.3333, A 0.000, B 0.000, C 0.000 }
gfCNCPoint4[23156] = {X 112.0487, Y 73.9693, Z -6.3333, A 0.000, B 0.000, C 0.000 }
gfCNCPoint4[23157] = {X 113.7647, Y 73.0876, Z -6.3333, A 0.000, B 0.000, C 0.000 }
gfCNCPoint4[23158] = {X 115.5404, Y 72.3332, Z -6.3333, A 0.000, B 0.000, C 0.000 }
gfCNCPoint4[23159] = {X 123.7265, Y 63.3438, Z -6.3333, A 0.000, B 0.000, C 0.000 }
gfCNCPoint4[23160] = {X 121.7844, Y 63.8620, Z -6.3333, A 0.000, B 0.000, C 0.000 }
gfCNCPoint4[23161] = {X 119.7989, Y 64.1752, Z -6.3333, A 0.000, B 0.000, C 0.000 }
gfCNCPoint4[23162] = {X 117.7916, Y 64.2800, Z -6.3333, A 0.000, B 0.000, C 0.000 }
gfCNCPoint4[23163] = {X 111.9185, Y 64.2800, Z -6.3333, A 0.000, B 0.000, C 0.000 }
gfCNCPoint4[23164] = {X 111.5741, Y 64.2769, Z -6.3333, A 0.000, B 0.000, C 0.000 }
gfCNCPoint4[23165] = {X 111.2299, Y 64.2677, Z -6.3333, A 0.000, B 0.000, C 0.000 }
gfCNCPoint4[23166] = {X 111.3156, Y 61.8692, Z -6.3333, A 0.000, B 0.000, C 0.000 }
gfCNCPoint4[23167] = {X 109.8654, Y 61.7547, Z -6.3333, A 0.000, B 0.000, C 0.000 }
gfCNCPoint4[23168] = {X 108.4304, Y 61.5157, Z -6.3333, A 0.000, B 0.000, C 0.000 }
gfCNCPoint4[23169] = {X 107.0213, Y 61.1540, Z -6.3333, A 0.000, B 0.000, C 0.000 }
gfCNCPoint4[23170] = {X 105.0907, Y 61.6173, Z -6.3333, A 0.000, B 0.000, C 0.000 }
gfCNCPoint4[23171] = {X 103.1191, Y 61.8506, Z -6.3333, A 0.000, B 0.000, C 0.000 }
gfCNCPoint4[23172] = {X 101.1337, Y 61.8509, Z -6.3333, A 0.000, B 0.000, C 0.000 }
gfCNCPoint4[23173] = {X 99.1620, Y 61.6181, Z -6.3333, A 0.000, B 0.000, C 0.000 }
gfCNCPoint4[23174] = {X 97.2313, Y 61.1553, Z -6.3333, A 0.000, B 0.000, C 0.000 }
gfCNCPoint4[23175] = {X 95.6267, Y 61.5566, Z -6.3333, A 0.000, B 0.000, C 0.000 }
gfCNCPoint4[23176] = {X 93.9906, Y 61.7990, Z -6.3333, A 0.000, B 0.000, C 0.000 }
gfCNCPoint4[23177] = {X 92.3385, Y 61.8800, Z -6.3333, A 0.000, B 0.000, C 0.000 }
gfCNCPoint4[23178] = {X 85.8951, Y 61.8800, Z -6.3333, A 0.000, B 0.000, C 0.000 }
gfCNCPoint4[23179] = {X 85.1609, Y 61.8640, Z -6.3333, A 0.000, B 0.000, C 0.000 }
gfCNCPoint4[23180] = {X 84.4280, Y 61.8161, Z -6.3333, A 0.000, B 0.000, C 0.000 }
gfCNCPoint4[23181] = {X 82.7246, Y 63.0692, Z -6.3333, A 0.000, B 0.000, C 0.000 }
gfCNCPoint4[23182] = {X 80.9073, Y 64.1504, Z -6.3333, A 0.000, B 0.000, C 0.000 }
gfCNCPoint4[23183] = {X 78.9932, Y 65.0494, Z -6.3333, A 0.000, B 0.000, C 0.000 }
gfCNCPoint4[23184] = {X 77.0007, Y 65.7577, Z -6.3333, A 0.000, B 0.000, C 0.000 }
gfCNCPoint4[23185] = {X 74.9487, Y 66.2685, Z -6.3333, A 0.000, B 0.000, C 0.000 }
gfCNCPoint4[23186] = {X 72.8566, Y 66.5769, Z -6.3333, A 0.000, B 0.000, C 0.000 }
gfCNCPoint4[23187] = {X 70.7445, Y 66.6800, Z -6.3333, A 0.000, B 0.000, C 0.000 }
gfCNCPoint4[23188] = {X 64.1851, Y 66.6800, Z -6.3333, A 0.000, B 0.000, C 0.000 }
gfCNCPoint4[23189] = {X 62.0576, Y 66.5754, Z -6.3333, A 0.000, B 0.000, C 0.000 }
gfCNCPoint4[23190] = {X 59.9505, Y 66.2624, Z -6.3333, A 0.000, B 0.000, C 0.000 }
gfCNCPoint4[23191] = {X 57.8844, Y 65.7442, Z -6.3333, A 0.000, B 0.000, C 0.000 }
gfCNCPoint4[23192] = {X 55.8790, Y 65.0258, Z -6.3333, A 0.000, B 0.000, C 0.000 }
gfCNCPoint4[23193] = {X 53.8737, Y 65.7442, Z -6.3333, A 0.000, B 0.000, C 0.000 }
gfCNCPoint4[23194] = {X 51.8075, Y 66.2624, Z -6.3333, A 0.000, B 0.000, C 0.000 }
gfCNCPoint4[23195] = {X 49.7005, Y 66.5754, Z -6.3333, A 0.000, B 0.000, C 0.000 }
gfCNCPoint4[23196] = {X 47.5729, Y 66.6800, Z -6.3333, A 0.000, B 0.000, C 0.000 }
gfCNCPoint4[23197] = {X 40.6393, Y 66.6800, Z -6.3333, A 0.000, B 0.000, C 0.000 }
gfCNCPoint4[23198] = {X 38.5451, Y 66.5786, Z -6.3333, A 0.000, B 0.000, C 0.000 }
gfCNCPoint4[23199] = {X 36.4705, Y 66.2754, Z -6.3333, A 0.000, B 0.000, C 0.000 }
gfCNCPoint4[23200] = {X 34.5045, Y 67.0020, Z -6.3333, A 0.000, B 0.000, C 0.000 }
gfCNCPoint4[23201] = {X 32.4863, Y 67.5678, Z -6.3333, A 0.000, B 0.000, C 0.000 }
gfCNCPoint4[23202] = {X 30.4290, Y 67.9694, Z -6.3333, A 0.000, B 0.000, C 0.000 }
gfCNCPoint4[23203] = {X 28.4166, Y 68.7664, Z -6.3333, A 0.000, B 0.000, C 0.000 }
gfCNCPoint4[23204] = {X 26.3723, Y 69.4774, Z -6.3333, A 0.000, B 0.000, C 0.000 }
gfCNCPoint4[23205] = {X 23.9562, Y 70.1962, Z -6.3333, A 0.000, B 0.000, C 0.000 }
gfCNCPoint4[23206] = {X 21.5034, Y 70.7769, Z -6.3333, A 0.000, B 0.000, C 0.000 }
gfCNCPoint4[23207] = {X 21.5034, Y 78.4951, Z -6.3333, A 0.000, B 0.000, C 0.000 }
gfCNCPoint4[23208] = {X 109.6713, Y 78.4951, Z -6.3333, A 0.000, B 0.000, C 0.000 }
gfCNCPoint4[23209] = {X 111.3424, Y 77.2337, Z -6.3333, A 0.000, B 0.000, C 0.000 }
gfCNCPoint4[23210] = {X 113.1168, Y 76.1223, Z -6.3333, A 0.000, B 0.000, C 0.000 }
gfCNCPoint4[23211] = {X 114.9810, Y 75.1692, Z -6.3333, A 0.000, B 0.000, C 0.000 }
gfCNCPoint4[23212] = {X 116.9210, Y 74.3817, Z -6.3333, A 0.000, B 0.000, C 0.000 }
gfCNCPoint4[23213] = {X 130.4107, Y 59.5681, Z -6.3333, A 0.000, B 0.000, C 0.000 }
gfCNCPoint4[23214] = {X 129.5276, Y 58.7530, Z -6.3333, A 0.000, B 0.000, C 0.000 }
gfCNCPoint4[23215] = {X 128.6970, Y 57.8844, Z -6.3333, A 0.000, B 0.000, C 0.000 }
gfCNCPoint4[23216] = {X 127.3927, Y 58.8836, Z -6.3333, A 0.000, B 0.000, C 0.000 }
gfCNCPoint4[23217] = {X 125.9974, Y 59.7512, Z -6.3333, A 0.000, B 0.000, C 0.000 }
gfCNCPoint4[23218] = {X 124.5245, Y 60.4791, Z -6.3333, A 0.000, B 0.000, C 0.000 }
gfCNCPoint4[23219] = {X 122.9877, Y 61.0604, Z -6.3333, A 0.000, B 0.000, C 0.000 }
gfCNCPoint4[23220] = {X 121.2873, Y 61.5141, Z -6.3333, A 0.000, B 0.000, C 0.000 }
gfCNCPoint4[23221] = {X 119.5490, Y 61.7883, Z -6.3333, A 0.000, B 0.000, C 0.000 }
gfCNCPoint4[23222] = {X 117.7916, Y 61.8800, Z -6.3333, A 0.000, B 0.000, C 0.000 }
gfCNCPoint4[23223] = {X 111.9185, Y 61.8800, Z -6.3333, A 0.000, B 0.000, C 0.000 }
gfCNCPoint4[23224] = {X 111.6170, Y 61.8773, Z -6.3333, A 0.000, B 0.000, C 0.000 }
gfCNCPoint4[23225] = {X 111.3156, Y 61.8692, Z -6.3333, A 0.000, B 0.000, C 0.000 }
gfCNCPoint4[23226] = {X 111.4013, Y 59.4708, Z -6.3333, A 0.000, B 0.000, C 0.000 }
gfCNCPoint4[23227] = {X 109.9149, Y 59.3407, Z -6.3333, A 0.000, B 0.000, C 0.000 }
gfCNCPoint4[23228] = {X 108.4496, Y 59.0584, Z -6.3333, A 0.000, B 0.000, C 0.000 }
gfCNCPoint4[23229] = {X 107.0213, Y 58.6267, Z -6.3333, A 0.000, B 0.000, C 0.000 }
gfCNCPoint4[23230] = {X 105.4260, Y 59.0985, Z -6.3333, A 0.000, B 0.000, C 0.000 }
gfCNCPoint4[23231] = {X 103.7872, Y 59.3842, Z -6.3333, A 0.000, B 0.000, C 0.000 }
gfCNCPoint4[23232] = {X 102.1264, Y 59.4800, Z -6.3333, A 0.000, B 0.000, C 0.000 }
gfCNCPoint4[23233] = {X 100.4656, Y 59.3847, Z -6.3333, A 0.000, B 0.000, C 0.000 }
gfCNCPoint4[23234] = {X 98.8267, Y 59.0996, Z -6.3333, A 0.000, B 0.000, C 0.000 }
gfCNCPoint4[23235] = {X 97.2313, Y 58.6283, Z -6.3333, A 0.000, B 0.000, C 0.000 }
gfCNCPoint4[23236] = {X 95.6367, Y 59.0994, Z -6.3333, A 0.000, B 0.000, C 0.000 }
gfCNCPoint4[23237] = {X 93.9986, Y 59.3845, Z -6.3333, A 0.000, B 0.000, C 0.000 }
gfCNCPoint4[23238] = {X 92.3385, Y 59.4800, Z -6.3333, A 0.000, B 0.000, C 0.000 }
gfCNCPoint4[23239] = {X 85.8951, Y 59.4800, Z -6.3333, A 0.000, B 0.000, C 0.000 }
gfCNCPoint4[23240] = {X 84.7780, Y 59.4368, Z -6.3333, A 0.000, B 0.000, C 0.000 }
gfCNCPoint4[23241] = {X 83.6677, Y 59.3077, Z -6.3333, A 0.000, B 0.000, C 0.000 }
gfCNCPoint4[23242] = {X 82.0978, Y 60.5827, Z -6.3333, A 0.000, B 0.000, C 0.000 }
gfCNCPoint4[23243] = {X 80.4031, Y 61.6862, Z -6.3333, A 0.000, B 0.000, C 0.000 }
gfCNCPoint4[23244] = {X 78.6021, Y 62.6061, Z -6.3333, A 0.000, B 0.000, C 0.000 }
gfCNCPoint4[23245] = {X 76.7146, Y 63.3324, Z -6.3333, A 0.000, B 0.000, C 0.000 }
gfCNCPoint4[23246] = {X 74.7614, Y 63.8569, Z -6.3333, A 0.000, B 0.000, C 0.000 }
gfCNCPoint4[23247] = {X 72.7640, Y 64.1739, Z -6.3333, A 0.000, B 0.000, C 0.000 }
gfCNCPoint4[23248] = {X 70.7445, Y 64.2800, Z -6.3333, A 0.000, B 0.000, C 0.000 }
gfCNCPoint4[23249] = {X 64.1851, Y 64.2800, Z -6.3333, A 0.000, B 0.000, C 0.000 }
gfCNCPoint4[23250] = {X 62.0428, Y 64.1606, Z -6.3333, A 0.000, B 0.000, C 0.000 }
gfCNCPoint4[23251] = {X 59.9269, Y 63.8039, Z -6.3333, A 0.000, B 0.000, C 0.000 }
gfCNCPoint4[23252] = {X 57.8638, Y 63.2143, Z -6.3333, A 0.000, B 0.000, C 0.000 }
gfCNCPoint4[23253] = {X 55.8790, Y 62.3991, Z -6.3333, A 0.000, B 0.000, C 0.000 }
gfCNCPoint4[23254] = {X 53.8942, Y 63.2143, Z -6.3333, A 0.000, B 0.000, C 0.000 }
gfCNCPoint4[23255] = {X 51.8311, Y 63.8039, Z -6.3333, A 0.000, B 0.000, C 0.000 }
gfCNCPoint4[23256] = {X 49.7153, Y 64.1606, Z -6.3333, A 0.000, B 0.000, C 0.000 }
gfCNCPoint4[23257] = {X 47.5729, Y 64.2800, Z -6.3333, A 0.000, B 0.000, C 0.000 }
gfCNCPoint4[23258] = {X 40.6393, Y 64.2800, Z -6.3333, A 0.000, B 0.000, C 0.000 }
gfCNCPoint4[23259] = {X 39.1551, Y 64.2228, Z -6.3333, A 0.000, B 0.000, C 0.000 }
gfCNCPoint4[23260] = {X 37.6797, Y 64.0515, Z -6.3333, A 0.000, B 0.000, C 0.000 }
gfCNCPoint4[23261] = {X 36.2218, Y 63.7671, Z -6.3333, A 0.000, B 0.000, C 0.000 }
gfCNCPoint4[23262] = {X 34.1355, Y 64.5951, Z -6.3333, A 0.000, B 0.000, C 0.000 }
gfCNCPoint4[23263] = {X 31.9799, Y 65.2213, Z -6.3333, A 0.000, B 0.000, C 0.000 }
gfCNCPoint4[23264] = {X 29.7746, Y 65.6399, Z -6.3333, A 0.000, B 0.000, C 0.000 }
gfCNCPoint4[23265] = {X 27.7188, Y 66.4651, Z -6.3333, A 0.000, B 0.000, C 0.000 }
gfCNCPoint4[23266] = {X 25.6275, Y 67.1959, Z -6.3333, A 0.000, B 0.000, C 0.000 }
gfCNCPoint4[23267] = {X 23.4819, Y 67.8386, Z -6.3333, A 0.000, B 0.000, C 0.000 }
gfCNCPoint4[23268] = {X 21.3051, Y 68.3660, Z -6.3333, A 0.000, B 0.000, C 0.000 }
gfCNCPoint4[23269] = {X 19.1034, Y 68.7768, Z -6.3333, A 0.000, B 0.000, C 0.000 }
gfCNCPoint4[23270] = {X 19.1034, Y 80.8951, Z -6.3333, A 0.000, B 0.000, C 0.000 }
gfCNCPoint4[23271] = {X 110.5596, Y 80.8951, Z -6.3333, A 0.000, B 0.000, C 0.000 }
gfCNCPoint4[23272] = {X 112.3066, Y 79.4904, Z -6.3333, A 0.000, B 0.000, C 0.000 }
gfCNCPoint4[23273] = {X 114.1893, Y 78.2736, Z -6.3333, A 0.000, B 0.000, C 0.000 }
gfCNCPoint4[23274] = {X 116.1877, Y 77.2577, Z -6.3333, A 0.000, B 0.000, C 0.000 }
gfCNCPoint4[23275] = {X 118.2802, Y 76.4536, Z -6.3333, A 0.000, B 0.000, C 0.000 }
gfCNCPoint4[23276] = {X 133.9629, Y 59.2319, Z -6.3333, A 0.000, B 0.000, C 0.000 }
gfCNCPoint4[23277] = {X 132.7152, Y 58.3545, Z -6.3333, A 0.000, B 0.000, C 0.000 }
gfCNCPoint4[23278] = {X 131.5519, Y 57.3680, Z -6.3333, A 0.000, B 0.000, C 0.000 }
gfCNCPoint4[23279] = {X 130.4824, Y 56.2805, Z -6.3333, A 0.000, B 0.000, C 0.000 }
gfCNCPoint4[23280] = {X 129.6655, Y 55.2988, Z -6.3333, A 0.000, B 0.000, C 0.000 }
gfCNCPoint4[23281] = {X 128.9251, Y 54.2582, Z -6.3333, A 0.000, B 0.000, C 0.000 }
gfCNCPoint4[23282] = {X 128.0750, Y 55.1942, Z -6.3333, A 0.000, B 0.000, C 0.000 }
gfCNCPoint4[23283] = {X 127.1464, Y 56.0525, Z -6.3333, A 0.000, B 0.000, C 0.000 }
gfCNCPoint4[23284] = {X 125.7915, Y 57.0695, Z -6.3333, A 0.000, B 0.000, C 0.000 }
gfCNCPoint4[23285] = {X 124.3270, Y 57.9212, Z -6.3333, A 0.000, B 0.000, C 0.000 }
gfCNCPoint4[23286] = {X 122.7731, Y 58.5961, Z -6.3333, A 0.000, B 0.000, C 0.000 }
gfCNCPoint4[23287] = {X 121.1510, Y 59.0849, Z -6.3333, A 0.000, B 0.000, C 0.000 }
gfCNCPoint4[23288] = {X 119.4828, Y 59.3809, Z -6.3333, A 0.000, B 0.000, C 0.000 }
gfCNCPoint4[23289] = {X 117.7916, Y 59.4800, Z -6.3333, A 0.000, B 0.000, C 0.000 }
gfCNCPoint4[23290] = {X 111.9185, Y 59.4800, Z -6.3333, A 0.000, B 0.000, C 0.000 }
gfCNCPoint4[23291] = {X 111.6599, Y 59.4777, Z -6.3333, A 0.000, B 0.000, C 0.000 }
gfCNCPoint4[23292] = {X 111.4013, Y 59.4708, Z -6.3333, A 0.000, B 0.000, C 0.000 }
gfCNCPoint4[23293] = {X 111.4871, Y 57.0723, Z -6.3333, A 0.000, B 0.000, C 0.000 }
gfCNCPoint4[23294] = {X 109.9587, Y 56.9200, Z -6.3333, A 0.000, B 0.000, C 0.000 }
gfCNCPoint4[23295] = {X 108.4621, Y 56.5750, Z -6.3333, A 0.000, B 0.000, C 0.000 }
gfCNCPoint4[23296] = {X 107.0213, Y 56.0428, Z -6.3333, A 0.000, B 0.000, C 0.000 }
gfCNCPoint4[23297] = {X 105.4432, Y 56.6151, Z -6.3333, A 0.000, B 0.000, C 0.000 }
gfCNCPoint4[23298] = {X 103.8010, Y 56.9630, Z -6.3333, A 0.000, B 0.000, C 0.000 }
gfCNCPoint4[23299] = {X 102.1265, Y 57.0800, Z -6.3333, A 0.000, B 0.000, C 0.000 }
gfCNCPoint4[23300] = {X 100.4519, Y 56.9637, Z -6.3333, A 0.000, B 0.000, C 0.000 }
gfCNCPoint4[23301] = {X 98.8096, Y 56.6164, Z -6.3333, A 0.000, B 0.000, C 0.000 }
gfCNCPoint4[23302] = {X 97.2313, Y 56.0448, Z -6.3333, A 0.000, B 0.000, C 0.000 }
gfCNCPoint4[23303] = {X 95.6538, Y 56.6162, Z -6.3333, A 0.000, B 0.000, C 0.000 }
gfCNCPoint4[23304] = {X 94.0123, Y 56.9635, Z -6.3333, A 0.000, B 0.000, C 0.000 }
gfCNCPoint4[23305] = {X 92.3385, Y 57.0800, Z -6.3333, A 0.000, B 0.000, C 0.000 }
gfCNCPoint4[23306] = {X 85.8951, Y 57.0800, Z -6.3333, A 0.000, B 0.000, C 0.000 }
gfCNCPoint4[23307] = {X 84.3894, Y 56.9858, Z -6.3333, A 0.000, B 0.000, C 0.000 }
gfCNCPoint4[23308] = {X 82.9073, Y 56.7047, Z -6.3333, A 0.000, B 0.000, C 0.000 }
gfCNCPoint4[23309] = {X 81.4846, Y 58.0224, Z -6.3333, A 0.000, B 0.000, C 0.000 }
gfCNCPoint4[23310] = {X 79.9203, Y 59.1682, Z -6.3333, A 0.000, B 0.000, C 0.000 }
gfCNCPoint4[23311] = {X 78.2348, Y 60.1271, Z -6.3333, A 0.000, B 0.000, C 0.000 }
gfCNCPoint4[23312] = {X 76.4504, Y 60.8864, Z -6.3333, A 0.000, B 0.000, C 0.000 }
gfCNCPoint4[23313] = {X 74.5908, Y 61.4359, Z -6.3333, A 0.000, B 0.000, C 0.000 }
gfCNCPoint4[23314] = {X 72.6804, Y 61.7686, Z -6.3333, A 0.000, B 0.000, C 0.000 }
gfCNCPoint4[23315] = {X 70.7445, Y 61.8800, Z -6.3333, A 0.000, B 0.000, C 0.000 }
gfCNCPoint4[23316] = {X 64.1851, Y 61.8800, Z -6.3333, A 0.000, B 0.000, C 0.000 }
gfCNCPoint4[23317] = {X 62.4514, Y 61.7907, Z -6.3333, A 0.000, B 0.000, C 0.000 }
gfCNCPoint4[23318] = {X 60.7359, Y 61.5238, Z -6.3333, A 0.000, B 0.000, C 0.000 }
gfCNCPoint4[23319] = {X 59.0570, Y 61.0822, Z -6.3333, A 0.000, B 0.000, C 0.000 }
gfCNCPoint4[23320] = {X 57.4323, Y 60.4704, Z -6.3333, A 0.000, B 0.000, C 0.000 }
gfCNCPoint4[23321] = {X 55.8790, Y 59.6950, Z -6.3333, A 0.000, B 0.000, C 0.000 }
gfCNCPoint4[23322] = {X 54.3258, Y 60.4704, Z -6.3333, A 0.000, B 0.000, C 0.000 }
gfCNCPoint4[23323] = {X 52.7011, Y 61.0822, Z -6.3333, A 0.000, B 0.000, C 0.000 }
gfCNCPoint4[23324] = {X 51.0221, Y 61.5238, Z -6.3333, A 0.000, B 0.000, C 0.000 }
gfCNCPoint4[23325] = {X 49.3067, Y 61.7907, Z -6.3333, A 0.000, B 0.000, C 0.000 }
gfCNCPoint4[23326] = {X 47.5729, Y 61.8800, Z -6.3333, A 0.000, B 0.000, C 0.000 }
gfCNCPoint4[23327] = {X 40.6393, Y 61.8800, Z -6.3333, A 0.000, B 0.000, C 0.000 }
gfCNCPoint4[23328] = {X 39.0680, Y 61.8067, Z -6.3333, A 0.000, B 0.000, C 0.000 }
gfCNCPoint4[23329] = {X 37.5103, Y 61.5875, Z -6.3333, A 0.000, B 0.000, C 0.000 }
gfCNCPoint4[23330] = {X 35.9798, Y 61.2242, Z -6.3333, A 0.000, B 0.000, C 0.000 }
gfCNCPoint4[23331] = {X 34.3392, Y 61.9608, Z -6.3333, A 0.000, B 0.000, C 0.000 }
gfCNCPoint4[23332] = {X 32.6421, Y 62.5559, Z -6.3333, A 0.000, B 0.000, C 0.000 }
gfCNCPoint4[23333] = {X 30.9007, Y 63.0050, Z -6.3333, A 0.000, B 0.000, C 0.000 }
gfCNCPoint4[23334] = {X 29.1275, Y 63.3051, Z -6.3333, A 0.000, B 0.000, C 0.000 }
gfCNCPoint4[23335] = {X 27.0248, Y 64.1618, Z -6.3333, A 0.000, B 0.000, C 0.000 }
gfCNCPoint4[23336] = {X 24.8827, Y 64.9144, Z -6.3333, A 0.000, B 0.000, C 0.000 }
gfCNCPoint4[23337] = {X 22.1999, Y 65.6932, Z -6.3333, A 0.000, B 0.000, C 0.000 }
gfCNCPoint4[23338] = {X 19.4690, Y 66.2812, Z -6.3333, A 0.000, B 0.000, C 0.000 }
gfCNCPoint4[23339] = {X 16.7034, Y 66.6753, Z -6.3333, A 0.000, B 0.000, C 0.000 }
gfCNCPoint4[23340] = {X 16.7034, Y 83.2951, Z -6.3333, A 0.000, B 0.000, C 0.000 }
gfCNCPoint4[23341] = {X 111.5062, Y 83.2951, Z -6.3333, A 0.000, B 0.000, C 0.000 }
gfCNCPoint4[23342] = {X 112.9247, Y 82.0358, Z -6.3333, A 0.000, B 0.000, C 0.000 }
gfCNCPoint4[23343] = {X 114.4600, Y 80.9220, Z -6.3333, A 0.000, B 0.000, C 0.000 }
gfCNCPoint4[23344] = {X 116.0974, Y 79.9644, Z -6.3333, A 0.000, B 0.000, C 0.000 }
gfCNCPoint4[23345] = {X 117.8209, Y 79.1724, Z -6.3333, A 0.000, B 0.000, C 0.000 }
gfCNCPoint4[23346] = {X 119.6140, Y 78.5535, Z -6.3333, A 0.000, B 0.000, C 0.000 }
gfCNCPoint4[23347] = {X 137.8566, Y 58.5206, Z -6.3333, A 0.000, B 0.000, C 0.000 }
gfCNCPoint4[23348] = {X 136.5219, Y 57.9302, Z -6.3333, A 0.000, B 0.000, C 0.000 }
gfCNCPoint4[23349] = {X 135.2534, Y 57.2084, Z -6.3333, A 0.000, B 0.000, C 0.000 }
gfCNCPoint4[23350] = {X 134.0096, Y 56.3194, Z -6.3333, A 0.000, B 0.000, C 0.000 }
gfCNCPoint4[23351] = {X 132.8665, Y 55.3043, Z -6.3333, A 0.000, B 0.000, C 0.000 }
gfCNCPoint4[23352] = {X 131.8368, Y 54.1742, Z -6.3333, A 0.000, B 0.000, C 0.000 }
gfCNCPoint4[23353] = {X 130.9319, Y 52.9419, Z -6.3333, A 0.000, B 0.000, C 0.000 }
gfCNCPoint4[23354] = {X 130.2147, Y 51.7225, Z -6.3333, A 0.000, B 0.000, C 0.000 }
gfCNCPoint4[23355] = {X 129.6199, Y 50.4390, Z -6.3333, A 0.000, B 0.000, C 0.000 }
gfCNCPoint4[23356] = {X 129.1532, Y 49.1035, Z -6.3333, A 0.000, B 0.000, C 0.000 }
gfCNCPoint4[23357] = {X 128.6036, Y 50.3877, Z -6.3333, A 0.000, B 0.000, C 0.000 }
gfCNCPoint4[23358] = {X 127.9093, Y 51.5998, Z -6.3333, A 0.000, B 0.000, C 0.000 }
gfCNCPoint4[23359] = {X 127.0798, Y 52.7237, Z -6.3333, A 0.000, B 0.000, C 0.000 }
gfCNCPoint4[23360] = {X 126.0417, Y 53.8239, Z -6.3333, A 0.000, B 0.000, C 0.000 }
gfCNCPoint4[23361] = {X 124.8743, Y 54.7858, Z -6.3333, A 0.000, B 0.000, C 0.000 }
gfCNCPoint4[23362] = {X 123.5958, Y 55.5942, Z -6.3333, A 0.000, B 0.000, C 0.000 }
gfCNCPoint4[23363] = {X 122.2263, Y 56.2365, Z -6.3333, A 0.000, B 0.000, C 0.000 }
gfCNCPoint4[23364] = {X 120.7872, Y 56.7027, Z -6.3333, A 0.000, B 0.000, C 0.000 }
gfCNCPoint4[23365] = {X 119.3012, Y 56.9853, Z -6.3333, A 0.000, B 0.000, C 0.000 }
gfCNCPoint4[23366] = {X 117.7916, Y 57.0800, Z -6.3333, A 0.000, B 0.000, C 0.000 }
gfCNCPoint4[23367] = {X 111.9185, Y 57.0800, Z -6.3333, A 0.000, B 0.000, C 0.000 }
gfCNCPoint4[23368] = {X 111.7027, Y 57.0781, Z -6.3333, A 0.000, B 0.000, C 0.000 }
gfCNCPoint4[23369] = {X 111.4871, Y 57.0723, Z -6.3333, A 0.000, B 0.000, C 0.000 }
gfCNCPoint4[23370] = {X 111.5728, Y 54.6738, Z -6.3333, A 0.000, B 0.000, C 0.000 }
gfCNCPoint4[23371] = {X 110.3820, Y 54.5573, Z -6.3333, A 0.000, B 0.000, C 0.000 }
gfCNCPoint4[23372] = {X 109.2147, Y 54.2947, Z -6.3333, A 0.000, B 0.000, C 0.000 }
gfCNCPoint4[23373] = {X 108.0887, Y 53.8902, Z -6.3333, A 0.000, B 0.000, C 0.000 }
gfCNCPoint4[23374] = {X 107.0213, Y 53.3498, Z -6.3333, A 0.000, B 0.000, C 0.000 }
gfCNCPoint4[23375] = {X 106.6480, Y 53.5578, Z -6.3333, A 0.000, B 0.000, C 0.000 }
gfCNCPoint4[23376] = {X 106.2658, Y 53.7492, Z -6.3333, A 0.000, B 0.000, C 0.000 }
gfCNCPoint4[23377] = {X 105.0149, Y 54.2383, Z -6.3333, A 0.000, B 0.000, C 0.000 }
gfCNCPoint4[23378] = {X 103.7084, Y 54.5495, Z -6.3333, A 0.000, B 0.000, C 0.000 }
gfCNCPoint4[23379] = {X 102.3713, Y 54.6768, Z -6.3333, A 0.000, B 0.000, C 0.000 }
gfCNCPoint4[23380] = {X 101.0295, Y 54.6179, Z -6.3333, A 0.000, B 0.000, C 0.000 }
gfCNCPoint4[23381] = {X 99.7088, Y 54.3738, Z -6.3333, A 0.000, B 0.000, C 0.000 }
gfCNCPoint4[23382] = {X 98.4345, Y 53.9493, Z -6.3333, A 0.000, B 0.000, C 0.000 }
gfCNCPoint4[23383] = {X 97.2313, Y 53.3524, Z -6.3333, A 0.000, B 0.000, C 0.000 }
gfCNCPoint4[23384] = {X 96.0852, Y 53.9255, Z -6.3333, A 0.000, B 0.000, C 0.000 }
gfCNCPoint4[23385] = {X 94.8734, Y 54.3422, Z -6.3333, A 0.000, B 0.000, C 0.000 }
gfCNCPoint4[23386] = {X 93.6172, Y 54.5952, Z -6.3333, A 0.000, B 0.000, C 0.000 }
gfCNCPoint4[23387] = {X 92.3385, Y 54.6800, Z -6.3333, A 0.000, B 0.000, C 0.000 }
gfCNCPoint4[23388] = {X 85.8951, Y 54.6800, Z -6.3333, A 0.000, B 0.000, C 0.000 }
gfCNCPoint4[23389] = {X 84.6159, Y 54.5951, Z -6.3333, A 0.000, B 0.000, C 0.000 }
gfCNCPoint4[23390] = {X 83.3592, Y 54.3419, Z -6.3333, A 0.000, B 0.000, C 0.000 }
gfCNCPoint4[23391] = {X 82.1469, Y 53.9249, Z -6.3333, A 0.000, B 0.000, C 0.000 }
gfCNCPoint4[23392] = {X 81.0644, Y 55.1572, Z -6.3333, A 0.000, B 0.000, C 0.000 }
gfCNCPoint4[23393] = {X 79.8495, Y 56.2591, Z -6.3333, A 0.000, B 0.000, C 0.000 }
gfCNCPoint4[23394] = {X 78.5178, Y 57.2166, Z -6.3333, A 0.000, B 0.000, C 0.000 }
gfCNCPoint4[23395] = {X 77.0863, Y 58.0174, Z -6.3333, A 0.000, B 0.000, C 0.000 }
gfCNCPoint4[23396] = {X 75.5734, Y 58.6511, Z -6.3333, A 0.000, B 0.000, C 0.000 }
gfCNCPoint4[23397] = {X 73.9986, Y 59.1096, Z -6.3333, A 0.000, B 0.000, C 0.000 }
gfCNCPoint4[23398] = {X 72.3820, Y 59.3871, Z -6.3333, A 0.000, B 0.000, C 0.000 }
gfCNCPoint4[23399] = {X 70.7445, Y 59.4800, Z -6.3333, A 0.000, B 0.000, C 0.000 }
gfCNCPoint4[23400] = {X 64.1851, Y 59.4800, Z -6.3333, A 0.000, B 0.000, C 0.000 }
gfCNCPoint4[23401] = {X 62.4203, Y 59.3720, Z -6.3333, A 0.000, B 0.000, C 0.000 }
gfCNCPoint4[23402] = {X 60.6818, Y 59.0498, Z -6.3333, A 0.000, B 0.000, C 0.000 }
gfCNCPoint4[23403] = {X 58.9955, Y 58.5181, Z -6.3333, A 0.000, B 0.000, C 0.000 }
gfCNCPoint4[23404] = {X 57.3866, Y 57.7848, Z -6.3333, A 0.000, B 0.000, C 0.000 }
gfCNCPoint4[23405] = {X 55.8790, Y 56.8608, Z -6.3333, A 0.000, B 0.000, C 0.000 }
gfCNCPoint4[23406] = {X 54.3715, Y 57.7848, Z -6.3333, A 0.000, B 0.000, C 0.000 }
gfCNCPoint4[23407] = {X 52.7626, Y 58.5181, Z -6.3333, A 0.000, B 0.000, C 0.000 }
gfCNCPoint4[23408] = {X 51.0763, Y 59.0498, Z -6.3333, A 0.000, B 0.000, C 0.000 }
gfCNCPoint4[23409] = {X 49.3378, Y 59.3720, Z -6.3333, A 0.000, B 0.000, C 0.000 }
gfCNCPoint4[23410] = {X 47.5729, Y 59.4800, Z -6.3333, A 0.000, B 0.000, C 0.000 }
gfCNCPoint4[23411] = {X 40.6393, Y 59.4800, Z -6.3333, A 0.000, B 0.000, C 0.000 }
gfCNCPoint4[23412] = {X 38.9798, Y 59.3846, Z -6.3333, A 0.000, B 0.000, C 0.000 }
gfCNCPoint4[23413] = {X 37.3422, Y 59.0996, Z -6.3333, A 0.000, B 0.000, C 0.000 }
gfCNCPoint4[23414] = {X 35.7480, Y 58.6288, Z -6.3333, A 0.000, B 0.000, C 0.000 }
gfCNCPoint4[23415] = {X 34.0324, Y 59.4879, Z -6.3333, A 0.000, B 0.000, C 0.000 }
gfCNCPoint4[23416] = {X 32.2383, Y 60.1677, Z -6.3333, A 0.000, B 0.000, C 0.000 }
gfCNCPoint4[23417] = {X 30.3843, Y 60.6612, Z -6.3333, A 0.000, B 0.000, C 0.000 }
gfCNCPoint4[23418] = {X 28.4896, Y 60.9633, Z -6.3333, A 0.000, B 0.000, C 0.000 }
gfCNCPoint4[23419] = {X 26.3359, Y 61.8559, Z -6.3333, A 0.000, B 0.000, C 0.000 }
gfCNCPoint4[23420] = {X 24.1379, Y 62.6329, Z -6.3333, A 0.000, B 0.000, C 0.000 }
gfCNCPoint4[23421] = {X 21.7309, Y 63.3361, Z -6.3333, A 0.000, B 0.000, C 0.000 }
gfCNCPoint4[23422] = {X 19.2821, Y 63.8758, Z -6.3333, A 0.000, B 0.000, C 0.000 }
gfCNCPoint4[23423] = {X 16.8025, Y 64.2494, Z -6.3333, A 0.000, B 0.000, C 0.000 }
gfCNCPoint4[23424] = {X 14.3034, Y 64.4552, Z -6.3333, A 0.000, B 0.000, C 0.000 }
gfCNCPoint4[23425] = {X 14.3034, Y 85.6951, Z -6.3333, A 0.000, B 0.000, C 0.000 }
gfCNCPoint4[23426] = {X 112.5245, Y 85.6951, Z -6.3333, A 0.000, B 0.000, C 0.000 }
gfCNCPoint4[23427] = {X 113.9432, Y 84.3113, Z -6.3333, A 0.000, B 0.000, C 0.000 }
gfCNCPoint4[23428] = {X 115.5143, Y 83.1032, Z -6.3333, A 0.000, B 0.000, C 0.000 }
gfCNCPoint4[23429] = {X 117.2162, Y 82.0877, Z -6.3333, A 0.000, B 0.000, C 0.000 }
gfCNCPoint4[23430] = {X 119.0254, Y 81.2786, Z -6.3333, A 0.000, B 0.000, C 0.000 }
gfCNCPoint4[23431] = {X 120.9170, Y 80.6872, Z -6.3333, A 0.000, B 0.000, C 0.000 }
gfCNCPoint4[23432] = {X 142.4286, Y 57.0645, Z -6.3333, A 0.000, B 0.000, C 0.000 }
gfCNCPoint4[23433] = {X 141.1657, Y 56.9338, Z -6.3333, A 0.000, B 0.000, C 0.000 }
gfCNCPoint4[23434] = {X 139.9235, Y 56.6712, Z -6.3333, A 0.000, B 0.000, C 0.000 }
gfCNCPoint4[23435] = {X 138.7157, Y 56.2796, Z -6.3333, A 0.000, B 0.000, C 0.000 }
gfCNCPoint4[23436] = {X 137.2787, Y 55.6178, Z -6.3333, A 0.000, B 0.000, C 0.000 }
gfCNCPoint4[23437] = {X 135.9405, Y 54.7739, Z -6.3333, A 0.000, B 0.000, C 0.000 }
gfCNCPoint4[23438] = {X 134.7241, Y 53.7624, Z -6.3333, A 0.000, B 0.000, C 0.000 }
gfCNCPoint4[23439] = {X 133.6504, Y 52.6005, Z -6.3333, A 0.000, B 0.000, C 0.000 }
gfCNCPoint4[23440] = {X 132.7376, Y 51.3083, Z -6.3333, A 0.000, B 0.000, C 0.000 }
gfCNCPoint4[23441] = {X 132.0016, Y 49.9080, Z -6.3333, A 0.000, B 0.000, C 0.000 }
gfCNCPoint4[23442] = {X 131.4549, Y 48.4234, Z -6.3333, A 0.000, B 0.000, C 0.000 }
gfCNCPoint4[23443] = {X 131.1845, Y 47.3200, Z -6.3333, A 0.000, B 0.000, C 0.000 }
gfCNCPoint4[23444] = {X 131.0190, Y 46.1961, Z -6.3333, A 0.000, B 0.000, C 0.000 }
gfCNCPoint4[23445] = {X 130.9598, Y 45.0616, Z -6.3333, A 0.000, B 0.000, C 0.000 }
gfCNCPoint4[23446] = {X 130.9601, Y 44.0978, Z -6.3333, A 0.000, B 0.000, C 0.000 }
gfCNCPoint4[23447] = {X 131.0921, Y 42.4244, Z -6.3333, A 0.000, B 0.000, C 0.000 }
gfCNCPoint4[23448] = {X 131.4548, Y 40.7854, Z -6.3333, A 0.000, B 0.000, C 0.000 }
gfCNCPoint4[23449] = {X 133.7565, Y 41.4655, Z -6.3333, A 0.000, B 0.000, C 0.000 }
gfCNCPoint4[23450] = {X 134.2330, Y 40.1906, Z -6.3333, A 0.000, B 0.000, C 0.000 }
gfCNCPoint4[23451] = {X 134.8836, Y 38.9952, Z -6.3333, A 0.000, B 0.000, C 0.000 }
gfCNCPoint4[23452] = {X 134.8836, Y 27.0854, Z -6.3333, A 0.000, B 0.000, C 0.000 }
gfCNCPoint4[23453] = {X 134.3931, Y 27.1259, Z -6.3333, A 0.000, B 0.000, C 0.000 }
gfCNCPoint4[23454] = {X 133.9011, Y 27.1414, Z -6.3333, A 0.000, B 0.000, C 0.000 }
gfCNCPoint4[23455] = {X 133.2006, Y 27.1415, Z -6.3333, A 0.000, B 0.000, C 0.000 }
gfCNCPoint4[23456] = {X 131.9567, Y 27.0613, Z -6.3333, A 0.000, B 0.000, C 0.000 }
gfCNCPoint4[23457] = {X 130.7334, Y 26.8218, Z -6.3333, A 0.000, B 0.000, C 0.000 }
gfCNCPoint4[23458] = {X 129.5511, Y 26.4272, Z -6.3333, A 0.000, B 0.000, C 0.000 }
gfCNCPoint4[23459] = {X 128.4292, Y 25.8839, Z -6.3333, A 0.000, B 0.000, C 0.000 }
gfCNCPoint4[23460] = {X 127.3865, Y 25.2009, Z -6.3333, A 0.000, B 0.000, C 0.000 }
gfCNCPoint4[23461] = {X 126.3458, Y 24.2963, Z -6.3333, A 0.000, B 0.000, C 0.000 }
gfCNCPoint4[23462] = {X 125.4443, Y 23.2530, Z -6.3333, A 0.000, B 0.000, C 0.000 }
gfCNCPoint4[23463] = {X 124.7001, Y 22.0922, Z -6.3333, A 0.000, B 0.000, C 0.000 }
gfCNCPoint4[23464] = {X 124.1284, Y 20.8375, Z -6.3333, A 0.000, B 0.000, C 0.000 }
gfCNCPoint4[23465] = {X 123.7408, Y 19.5142, Z -6.3333, A 0.000, B 0.000, C 0.000 }
gfCNCPoint4[23466] = {X 123.5451, Y 18.1493, Z -6.3333, A 0.000, B 0.000, C 0.000 }
gfCNCPoint4[23467] = {X 123.5447, Y 39.7478, Z -6.3333, A 0.000, B 0.000, C 0.000 }
gfCNCPoint4[23468] = {X 124.1929, Y 40.7417, Z -6.3333, A 0.000, B 0.000, C 0.000 }
gfCNCPoint4[23469] = {X 124.6711, Y 41.8276, Z -6.3333, A 0.000, B 0.000, C 0.000 }
gfCNCPoint4[23470] = {X 124.9666, Y 42.9768, Z -6.3333, A 0.000, B 0.000, C 0.000 }
gfCNCPoint4[23471] = {X 125.0714, Y 44.1587, Z -6.3333, A 0.000, B 0.000, C 0.000 }
gfCNCPoint4[23472] = {X 125.0716, Y 45.0000, Z -6.3333, A 0.000, B 0.000, C 0.000 }
gfCNCPoint4[23473] = {X 124.9610, Y 46.2642, Z -6.3333, A 0.000, B 0.000, C 0.000 }
gfCNCPoint4[23474] = {X 124.6325, Y 47.4899, Z -6.3333, A 0.000, B 0.000, C 0.000 }
gfCNCPoint4[23475] = {X 124.0962, Y 48.6400, Z -6.3333, A 0.000, B 0.000, C 0.000 }
gfCNCPoint4[23476] = {X 123.3684, Y 49.6795, Z -6.3333, A 0.000, B 0.000, C 0.000 }
gfCNCPoint4[23477] = {X 122.4711, Y 50.5768, Z -6.3333, A 0.000, B 0.000, C 0.000 }
gfCNCPoint4[23478] = {X 121.4316, Y 51.3047, Z -6.3333, A 0.000, B 0.000, C 0.000 }
gfCNCPoint4[23479] = {X 120.2815, Y 51.8410, Z -6.3333, A 0.000, B 0.000, C 0.000 }
gfCNCPoint4[23480] = {X 119.0557, Y 52.1694, Z -6.3333, A 0.000, B 0.000, C 0.000 }
gfCNCPoint4[23481] = {X 117.7916, Y 52.2800, Z -6.3333, A 0.000, B 0.000, C 0.000 }
gfCNCPoint4[23482] = {X 111.9185, Y 52.2800, Z -6.3333, A 0.000, B 0.000, C 0.000 }
gfCNCPoint4[23483] = {X 110.8481, Y 52.2009, Z -6.3333, A 0.000, B 0.000, C 0.000 }
gfCNCPoint4[23484] = {X 109.8009, Y 51.9652, Z -6.3333, A 0.000, B 0.000, C 0.000 }
gfCNCPoint4[23485] = {X 108.7998, Y 51.5782, Z -6.3333, A 0.000, B 0.000, C 0.000 }
gfCNCPoint4[23486] = {X 107.8665, Y 51.0481, Z -6.3333, A 0.000, B 0.000, C 0.000 }
gfCNCPoint4[23487] = {X 107.0213, Y 50.3866, Z -6.3333, A 0.000, B 0.000, C 0.000 }
gfCNCPoint4[23488] = {X 106.1743, Y 51.0493, Z -6.3333, A 0.000, B 0.000, C 0.000 }
gfCNCPoint4[23489] = {X 105.2389, Y 51.5800, Z -6.3333, A 0.000, B 0.000, C 0.000 }
gfCNCPoint4[23490] = {X 104.0917, Y 52.0091, Z -6.3333, A 0.000, B 0.000, C 0.000 }
gfCNCPoint4[23491] = {X 102.8887, Y 52.2397, Z -6.3333, A 0.000, B 0.000, C 0.000 }
gfCNCPoint4[23492] = {X 101.6641, Y 52.2655, Z -6.3333, A 0.000, B 0.000, C 0.000 }
gfCNCPoint4[23493] = {X 100.4526, Y 52.0855, Z -6.3333, A 0.000, B 0.000, C 0.000 }
gfCNCPoint4[23494] = {X 99.2883, Y 51.7050, Z -6.3333, A 0.000, B 0.000, C 0.000 }
gfCNCPoint4[23495] = {X 98.2043, Y 51.1347, Z -6.3333, A 0.000, B 0.000, C 0.000 }
gfCNCPoint4[23496] = {X 97.2313, Y 50.3907, Z -6.3333, A 0.000, B 0.000, C 0.000 }
gfCNCPoint4[23497] = {X 96.3865, Y 51.0508, Z -6.3333, A 0.000, B 0.000, C 0.000 }
gfCNCPoint4[23498] = {X 95.4539, Y 51.5797, Z -6.3333, A 0.000, B 0.000, C 0.000 }
gfCNCPoint4[23499] = {X 94.4538, Y 51.9659, Z -6.3333, A 0.000, B 0.000, C 0.000 }
gfCNCPoint4[23500] = {X 93.4078, Y 52.2011, Z -6.3333, A 0.000, B 0.000, C 0.000 }
gfCNCPoint4[23501] = {X 92.3385, Y 52.2800, Z -6.3333, A 0.000, B 0.000, C 0.000 }
gfCNCPoint4[23502] = {X 85.8951, Y 52.2800, Z -6.3333, A 0.000, B 0.000, C 0.000 }
gfCNCPoint4[23503] = {X 84.6852, Y 52.1788, Z -6.3333, A 0.000, B 0.000, C 0.000 }
gfCNCPoint4[23504] = {X 83.5090, Y 51.8779, Z -6.3333, A 0.000, B 0.000, C 0.000 }
gfCNCPoint4[23505] = {X 82.3992, Y 51.3857, Z -6.3333, A 0.000, B 0.000, C 0.000 }
gfCNCPoint4[23506] = {X 81.3866, Y 50.7159, Z -6.3333, A 0.000, B 0.000, C 0.000 }
gfCNCPoint4[23507] = {X 80.5223, Y 52.0937, Z -6.3333, A 0.000, B 0.000, C 0.000 }
gfCNCPoint4[23508] = {X 79.4808, Y 53.3429, Z -6.3333, A 0.000, B 0.000, C 0.000 }
gfCNCPoint4[23509] = {X 78.2809, Y 54.4408, Z -6.3333, A 0.000, B 0.000, C 0.000 }
gfCNCPoint4[23510] = {X 76.9444, Y 55.3676, Z -6.3333, A 0.000, B 0.000, C 0.000 }
gfCNCPoint4[23511] = {X 75.4955, Y 56.1065, Z -6.3333, A 0.000, B 0.000, C 0.000 }
gfCNCPoint4[23512] = {X 73.9605, Y 56.6440, Z -6.3333, A 0.000, B 0.000, C 0.000 }
gfCNCPoint4[23513] = {X 72.3672, Y 56.9705, Z -6.3333, A 0.000, B 0.000, C 0.000 }
gfCNCPoint4[23514] = {X 70.7445, Y 57.0800, Z -6.3333, A 0.000, B 0.000, C 0.000 }
gfCNCPoint4[23515] = {X 64.1851, Y 57.0800, Z -6.3333, A 0.000, B 0.000, C 0.000 }
gfCNCPoint4[23516] = {X 62.6628, Y 56.9837, Z -6.3333, A 0.000, B 0.000, C 0.000 }
gfCNCPoint4[23517] = {X 61.1646, Y 56.6963, Z -6.3333, A 0.000, B 0.000, C 0.000 }
gfCNCPoint4[23518] = {X 59.7147, Y 56.2224, Z -6.3333, A 0.000, B 0.000, C 0.000 }
gfCNCPoint4[23519] = {X 58.3360, Y 55.5695, Z -6.3333, A 0.000, B 0.000, C 0.000 }
gfCNCPoint4[23520] = {X 57.0507, Y 54.7481, Z -6.3333, A 0.000, B 0.000, C 0.000 }
gfCNCPoint4[23521] = {X 55.8790, Y 53.7713, Z -6.3333, A 0.000, B 0.000, C 0.000 }
gfCNCPoint4[23522] = {X 54.7074, Y 54.7481, Z -6.3333, A 0.000, B 0.000, C 0.000 }
gfCNCPoint4[23523] = {X 53.4220, Y 55.5695, Z -6.3333, A 0.000, B 0.000, C 0.000 }
gfCNCPoint4[23524] = {X 52.0434, Y 56.2224, Z -6.3333, A 0.000, B 0.000, C 0.000 }
gfCNCPoint4[23525] = {X 50.5934, Y 56.6963, Z -6.3333, A 0.000, B 0.000, C 0.000 }
gfCNCPoint4[23526] = {X 49.0953, Y 56.9837, Z -6.3333, A 0.000, B 0.000, C 0.000 }
gfCNCPoint4[23527] = {X 47.5729, Y 57.0800, Z -6.3333, A 0.000, B 0.000, C 0.000 }
gfCNCPoint4[23528] = {X 40.6393, Y 57.0800, Z -6.3333, A 0.000, B 0.000, C 0.000 }
gfCNCPoint4[23529] = {X 39.3238, Y 57.0082, Z -6.3333, A 0.000, B 0.000, C 0.000 }
gfCNCPoint4[23530] = {X 38.0240, Y 56.7935, Z -6.3333, A 0.000, B 0.000, C 0.000 }
gfCNCPoint4[23531] = {X 36.7553, Y 56.4386, Z -6.3333, A 0.000, B 0.000, C 0.000 }
gfCNCPoint4[23532] = {X 35.5328, Y 55.9476, Z -6.3333, A 0.000, B 0.000, C 0.000 }
gfCNCPoint4[23533] = {X 34.1213, Y 56.7829, Z -6.3333, A 0.000, B 0.000, C 0.000 }
gfCNCPoint4[23534] = {X 32.6336, Y 57.4732, Z -6.3333, A 0.000, B 0.000, C 0.000 }
gfCNCPoint4[23535] = {X 31.0844, Y 58.0116, Z -6.3333, A 0.000, B 0.000, C 0.000 }
gfCNCPoint4[23536] = {X 29.4891, Y 58.3926, Z -6.3333, A 0.000, B 0.000, C 0.000 }
gfCNCPoint4[23537] = {X 27.8639, Y 58.6125, Z -6.3333, A 0.000, B 0.000, C 0.000 }
gfCNCPoint4[23538] = {X 25.6536, Y 59.5467, Z -6.3333, A 0.000, B 0.000, C 0.000 }
gfCNCPoint4[23539] = {X 23.3930, Y 60.3514, Z -6.3333, A 0.000, B 0.000, C 0.000 }
gfCNCPoint4[23540] = {X 21.1523, Y 61.0069, Z -6.3333, A 0.000, B 0.000, C 0.000 }
gfCNCPoint4[23541] = {X 18.8726, Y 61.5108, Z -6.3333, A 0.000, B 0.000, C 0.000 }
gfCNCPoint4[23542] = {X 16.5643, Y 61.8609, Z -6.3333, A 0.000, B 0.000, C 0.000 }
gfCNCPoint4[23543] = {X 14.2377, Y 62.0555, Z -6.3333, A 0.000, B 0.000, C 0.000 }
gfCNCPoint4[23544] = {X 11.9034, Y 62.0939, Z -6.3333, A 0.000, B 0.000, C 0.000 }
gfCNCPoint4[23545] = {X 11.9034, Y 88.0951, Z -6.3333, A 0.000, B 0.000, C 0.000 }
gfCNCPoint4[23546] = {X 113.6336, Y 88.0951, Z -6.3333, A 0.000, B 0.000, C 0.000 }
gfCNCPoint4[23547] = {X 114.7667, Y 86.8215, Z -6.3333, A 0.000, B 0.000, C 0.000 }
gfCNCPoint4[23548] = {X 116.0415, Y 85.6898, Z -6.3333, A 0.000, B 0.000, C 0.000 }
gfCNCPoint4[23549] = {X 117.4406, Y 84.7158, Z -6.3333, A 0.000, B 0.000, C 0.000 }
gfCNCPoint4[23550] = {X 118.9444, Y 83.9130, Z -6.3333, A 0.000, B 0.000, C 0.000 }
gfCNCPoint4[23551] = {X 120.5321, Y 83.2925, Z -6.3333, A 0.000, B 0.000, C 0.000 }
gfCNCPoint4[23552] = {X 122.1818, Y 82.8628, Z -6.3333, A 0.000, B 0.000, C 0.000 }
gfCNCPoint4[23553] = {X 144.8180, Y 58.0052, Z -6.3333, A 0.000, B 0.000, C 0.000 }
gfCNCPoint4[23554] = {X 144.9144, Y 56.3314, Z -6.3333, A 0.000, B 0.000, C 0.000 }
gfCNCPoint4[23555] = {X 145.2037, Y 54.6800, Z -6.3333, A 0.000, B 0.000, C 0.000 }
gfCNCPoint4[23556] = {X 143.0396, Y 54.6800, Z -6.3333, A 0.000, B 0.000, C 0.000 }
gfCNCPoint4[23557] = {X 142.7947, Y 54.6769, Z -6.3333, A 0.000, B 0.000, C 0.000 }
gfCNCPoint4[23558] = {X 142.5500, Y 54.6676, Z -6.3333, A 0.000, B 0.000, C 0.000 }
gfCNCPoint4[23559] = {X 141.0970, Y 54.4831, Z -6.3333, A 0.000, B 0.000, C 0.000 }
gfCNCPoint4[23560] = {X 139.6885, Y 54.0814, Z -6.3333, A 0.000, B 0.000, C 0.000 }
gfCNCPoint4[23561] = {X 138.3568, Y 53.4719, Z -6.3333, A 0.000, B 0.000, C 0.000 }
gfCNCPoint4[23562] = {X 137.1322, Y 52.6684, Z -6.3333, A 0.000, B 0.000, C 0.000 }
gfCNCPoint4[23563] = {X 136.0429, Y 51.6894, Z -6.3333, A 0.000, B 0.000, C 0.000 }
gfCNCPoint4[23564] = {X 135.1137, Y 50.5572, Z -6.3333, A 0.000, B 0.000, C 0.000 }
gfCNCPoint4[23565] = {X 134.3660, Y 49.2978, Z -6.3333, A 0.000, B 0.000, C 0.000 }
gfCNCPoint4[23566] = {X 133.8169, Y 47.9400, Z -6.3333, A 0.000, B 0.000, C 0.000 }
gfCNCPoint4[23567] = {X 133.4789, Y 46.5150, Z -6.3333, A 0.000, B 0.000, C 0.000 }
gfCNCPoint4[23568] = {X 133.3598, Y 45.0552, Z -6.3333, A 0.000, B 0.000, C 0.000 }
gfCNCPoint4[23569] = {X 133.3601, Y 44.1104, Z -6.3333, A 0.000, B 0.000, C 0.000 }
gfCNCPoint4[23570] = {X 133.4665, Y 42.7742, Z -6.3333, A 0.000, B 0.000, C 0.000 }
gfCNCPoint4[23571] = {X 133.7565, Y 41.4655, Z -6.3333, A 0.000, B 0.000, C 0.000 }
gfCNCPoint4[23572] = {X 136.0581, Y 42.1457, Z -6.3333, A 0.000, B 0.000, C 0.000 }
gfCNCPoint4[23573] = {X 136.3664, Y 41.2990, Z -6.3333, A 0.000, B 0.000, C 0.000 }
gfCNCPoint4[23574] = {X 136.7770, Y 40.4969, Z -6.3333, A 0.000, B 0.000, C 0.000 }
gfCNCPoint4[23575] = {X 137.2836, Y 39.7516, Z -6.3333, A 0.000, B 0.000, C 0.000 }
gfCNCPoint4[23576] = {X 137.2836, Y 23.8768, Z -6.3333, A 0.000, B 0.000, C 0.000 }
gfCNCPoint4[23577] = {X 136.4352, Y 24.2641, Z -6.3333, A 0.000, B 0.000, C 0.000 }
gfCNCPoint4[23578] = {X 135.5443, Y 24.5398, Z -6.3333, A 0.000, B 0.000, C 0.000 }
gfCNCPoint4[23579] = {X 134.6254, Y 24.6993, Z -6.3333, A 0.000, B 0.000, C 0.000 }
gfCNCPoint4[23580] = {X 134.2595, Y 24.7296, Z -6.3333, A 0.000, B 0.000, C 0.000 }
gfCNCPoint4[23581] = {X 133.8926, Y 24.7414, Z -6.3333, A 0.000, B 0.000, C 0.000 }
gfCNCPoint4[23582] = {X 133.2006, Y 24.7415, Z -6.3333, A 0.000, B 0.000, C 0.000 }
gfCNCPoint4[23583] = {X 131.9932, Y 24.6407, Z -6.3333, A 0.000, B 0.000, C 0.000 }
gfCNCPoint4[23584] = {X 130.8191, Y 24.3410, Z -6.3333, A 0.000, B 0.000, C 0.000 }
gfCNCPoint4[23585] = {X 129.7111, Y 23.8507, Z -6.3333, A 0.000, B 0.000, C 0.000 }
gfCNCPoint4[23586] = {X 128.6997, Y 23.1834, Z -6.3333, A 0.000, B 0.000, C 0.000 }
gfCNCPoint4[23587] = {X 127.8130, Y 22.3576, Z -6.3333, A 0.000, B 0.000, C 0.000 }
gfCNCPoint4[23588] = {X 127.0756, Y 21.3962, Z -6.3333, A 0.000, B 0.000, C 0.000 }
gfCNCPoint4[23589] = {X 126.5078, Y 20.3258, Z -6.3333, A 0.000, B 0.000, C 0.000 }
gfCNCPoint4[23590] = {X 126.1254, Y 19.1761, Z -6.3333, A 0.000, B 0.000, C 0.000 }
gfCNCPoint4[23591] = {X 125.9390, Y 17.9788, Z -6.3333, A 0.000, B 0.000, C 0.000 }
gfCNCPoint4[23592] = {X 125.9252, Y 17.7203, Z -6.3333, A 0.000, B 0.000, C 0.000 }
gfCNCPoint4[23593] = {X 125.9206, Y 17.4615, Z -6.3333, A 0.000, B 0.000, C 0.000 }
gfCNCPoint4[23594] = {X 125.9206, Y 10.4835, Z -6.3333, A 0.000, B 0.000, C 0.000 }
gfCNCPoint4[23595] = {X 125.9372, Y 9.9931, Z -6.3333, A 0.000, B 0.000, C 0.000 }
gfCNCPoint4[23596] = {X 125.9867, Y 9.5049, Z -6.3333, A 0.000, B 0.000, C 0.000 }
gfCNCPoint4[23597] = {X 121.8686, Y 9.5049, Z -6.3333, A 0.000, B 0.000, C 0.000 }
gfCNCPoint4[23598] = {X 122.3090, Y 10.3410, Z -6.3333, A 0.000, B 0.000, C 0.000 }
gfCNCPoint4[23599] = {X 122.5801, Y 11.2463, Z -6.3333, A 0.000, B 0.000, C 0.000 }
gfCNCPoint4[23600] = {X 122.6716, Y 12.1868, Z -6.3333, A 0.000, B 0.000, C 0.000 }
gfCNCPoint4[23601] = {X 122.6714, Y 13.0237, Z -6.3333, A 0.000, B 0.000, C 0.000 }
gfCNCPoint4[23602] = {X 122.5640, Y 13.9968, Z -6.3333, A 0.000, B 0.000, C 0.000 }
gfCNCPoint4[23603] = {X 122.2647, Y 14.9289, Z -6.3333, A 0.000, B 0.000, C 0.000 }
gfCNCPoint4[23604] = {X 121.7853, Y 15.7825, Z -6.3333, A 0.000, B 0.000, C 0.000 }
gfCNCPoint4[23605] = {X 121.1451, Y 16.5232, Z -6.3333, A 0.000, B 0.000, C 0.000 }
gfCNCPoint4[23606] = {X 121.1447, Y 40.6632, Z -6.3333, A 0.000, B 0.000, C 0.000 }
gfCNCPoint4[23607] = {X 121.7858, Y 41.4051, Z -6.3333, A 0.000, B 0.000, C 0.000 }
gfCNCPoint4[23608] = {X 122.2657, Y 42.2602, Z -6.3333, A 0.000, B 0.000, C 0.000 }
gfCNCPoint4[23609] = {X 122.5649, Y 43.1940, Z -6.3333, A 0.000, B 0.000, C 0.000 }
gfCNCPoint4[23610] = {X 122.6714, Y 44.1688, Z -6.3333, A 0.000, B 0.000, C 0.000 }
gfCNCPoint4[23611] = {X 122.6716, Y 45.0000, Z -6.3333, A 0.000, B 0.000, C 0.000 }
gfCNCPoint4[23612] = {X 122.5778, Y 45.9520, Z -6.3333, A 0.000, B 0.000, C 0.000 }
gfCNCPoint4[23613] = {X 122.3001, Y 46.8675, Z -6.3333, A 0.000, B 0.000, C 0.000 }
gfCNCPoint4[23614] = {X 121.8491, Y 47.7112, Z -6.3333, A 0.000, B 0.000, C 0.000 }
gfCNCPoint4[23615] = {X 121.2423, Y 48.4507, Z -6.3333, A 0.000, B 0.000, C 0.000 }
gfCNCPoint4[23616] = {X 120.5028, Y 49.0576, Z -6.3333, A 0.000, B 0.000, C 0.000 }
gfCNCPoint4[23617] = {X 119.6591, Y 49.5085, Z -6.3333, A 0.000, B 0.000, C 0.000 }
gfCNCPoint4[23618] = {X 118.7436, Y 49.7862, Z -6.3333, A 0.000, B 0.000, C 0.000 }
gfCNCPoint4[23619] = {X 117.7916, Y 49.8800, Z -6.3333, A 0.000, B 0.000, C 0.000 }
gfCNCPoint4[23620] = {X 111.9185, Y 49.8800, Z -6.3333, A 0.000, B 0.000, C 0.000 }
gfCNCPoint4[23621] = {X 111.0234, Y 49.7972, Z -6.3333, A 0.000, B 0.000, C 0.000 }
gfCNCPoint4[23622] = {X 110.1587, Y 49.5517, Z -6.3333, A 0.000, B 0.000, C 0.000 }
gfCNCPoint4[23623] = {X 109.3537, Y 49.1517, Z -6.3333, A 0.000, B 0.000, C 0.000 }
gfCNCPoint4[23624] = {X 108.6357, Y 48.6108, Z -6.3333, A 0.000, B 0.000, C 0.000 }
gfCNCPoint4[23625] = {X 108.0714, Y 48.0024, Z -6.3333, A 0.000, B 0.000, C 0.000 }
gfCNCPoint4[23626] = {X 107.6183, Y 47.3071, Z -6.3333, A 0.000, B 0.000, C 0.000 }
gfCNCPoint4[23627] = {X 107.2895, Y 46.5451, Z -6.3333, A 0.000, B 0.000, C 0.000 }
gfCNCPoint4[23628] = {X 107.0947, Y 45.7384, Z -6.3333, A 0.000, B 0.000, C 0.000 }
gfCNCPoint4[23629] = {X 106.6287, Y 46.8768, Z -6.3333, A 0.000, B 0.000, C 0.000 }
gfCNCPoint4[23630] = {X 106.1131, Y 47.8110, Z -6.3333, A 0.000, B 0.000, C 0.000 }
gfCNCPoint4[23631] = {X 105.4068, Y 48.6108, Z -6.3333, A 0.000, B 0.000, C 0.000 }
gfCNCPoint4[23632] = {X 104.8391, Y 49.0550, Z -6.3333, A 0.000, B 0.000, C 0.000 }
gfCNCPoint4[23633] = {X 104.2121, Y 49.4107, Z -6.3333, A 0.000, B 0.000, C 0.000 }
gfCNCPoint4[23634] = {X 103.3106, Y 49.7335, Z -6.3333, A 0.000, B 0.000, C 0.000 }
gfCNCPoint4[23635] = {X 102.3635, Y 49.8741, Z -6.3333, A 0.000, B 0.000, C 0.000 }
gfCNCPoint4[23636] = {X 101.4071, Y 49.8271, Z -6.3333, A 0.000, B 0.000, C 0.000 }
gfCNCPoint4[23637] = {X 100.4784, Y 49.5941, Z -6.3333, A 0.000, B 0.000, C 0.000 }
gfCNCPoint4[23638] = {X 99.6130, Y 49.1844, Z -6.3333, A 0.000, B 0.000, C 0.000 }
gfCNCPoint4[23639] = {X 98.8443, Y 48.6135, Z -6.3333, A 0.000, B 0.000, C 0.000 }
gfCNCPoint4[23640] = {X 98.1362, Y 47.8127, Z -6.3333, A 0.000, B 0.000, C 0.000 }
gfCNCPoint4[23641] = {X 97.6194, Y 46.8769, Z -6.3333, A 0.000, B 0.000, C 0.000 }
gfCNCPoint4[23642] = {X 97.1600, Y 45.7536, Z -6.3333, A 0.000, B 0.000, C 0.000 }
gfCNCPoint4[23643] = {X 96.9635, Y 46.5570, Z -6.3333, A 0.000, B 0.000, C 0.000 }
gfCNCPoint4[23644] = {X 96.6342, Y 47.3156, Z -6.3333, A 0.000, B 0.000, C 0.000 }
gfCNCPoint4[23645] = {X 96.1814, Y 48.0078, Z -6.3333, A 0.000, B 0.000, C 0.000 }
gfCNCPoint4[23646] = {X 95.6183, Y 48.6135, Z -6.3333, A 0.000, B 0.000, C 0.000 }
gfCNCPoint4[23647] = {X 94.9007, Y 49.1533, Z -6.3333, A 0.000, B 0.000, C 0.000 }
gfCNCPoint4[23648] = {X 94.0964, Y 49.5524, Z -6.3333, A 0.000, B 0.000, C 0.000 }
gfCNCPoint4[23649] = {X 93.2326, Y 49.7974, Z -6.3333, A 0.000, B 0.000, C 0.000 }
gfCNCPoint4[23650] = {X 92.3385, Y 49.8800, Z -6.3333, A 0.000, B 0.000, C 0.000 }
gfCNCPoint4[23651] = {X 85.8951, Y 49.8800, Z -6.3333, A 0.000, B 0.000, C 0.000 }
gfCNCPoint4[23652] = {X 85.0841, Y 49.8121, Z -6.3333, A 0.000, B 0.000, C 0.000 }
gfCNCPoint4[23653] = {X 84.2956, Y 49.6104, Z -6.3333, A 0.000, B 0.000, C 0.000 }
gfCNCPoint4[23654] = {X 83.5517, Y 49.2805, Z -6.3333, A 0.000, B 0.000, C 0.000 }
gfCNCPoint4[23655] = {X 82.8729, Y 48.8316, Z -6.3333, A 0.000, B 0.000, C 0.000 }
gfCNCPoint4[23656] = {X 82.2391, Y 48.2324, Z -6.3333, A 0.000, B 0.000, C 0.000 }
gfCNCPoint4[23657] = {X 81.7221, Y 47.5300, Z -6.3333, A 0.000, B 0.000, C 0.000 }
gfCNCPoint4[23658] = {X 81.3384, Y 46.7467, Z -6.3333, A 0.000, B 0.000, C 0.000 }
gfCNCPoint4[23659] = {X 81.1002, Y 45.9077, Z -6.3333, A 0.000, B 0.000, C 0.000 }
gfCNCPoint4[23660] = {X 81.0152, Y 45.0397, Z -6.3333, A 0.000, B 0.000, C 0.000 }
gfCNCPoint4[23661] = {X 81.0151, Y 44.2042, Z -6.3333, A 0.000, B 0.000, C 0.000 }
gfCNCPoint4[23662] = {X 81.1195, Y 43.2203, Z -6.3333, A 0.000, B 0.000, C 0.000 }
gfCNCPoint4[23663] = {X 81.4180, Y 42.2770, Z -6.3333, A 0.000, B 0.000, C 0.000 }
gfCNCPoint4[23664] = {X 81.8987, Y 41.4121, Z -6.3333, A 0.000, B 0.000, C 0.000 }
gfCNCPoint4[23665] = {X 82.5422, Y 40.6606, Z -6.3333, A 0.000, B 0.000, C 0.000 }
gfCNCPoint4[23666] = {X 82.5419, Y 16.5235, Z -6.3333, A 0.000, B 0.000, C 0.000 }
gfCNCPoint4[23667] = {X 81.9010, Y 15.7819, Z -6.3333, A 0.000, B 0.000, C 0.000 }
gfCNCPoint4[23668] = {X 81.4213, Y 14.9273, Z -6.3333, A 0.000, B 0.000, C 0.000 }
gfCNCPoint4[23669] = {X 81.1220, Y 13.9939, Z -6.3333, A 0.000, B 0.000, C 0.000 }
gfCNCPoint4[23670] = {X 81.0153, Y 13.0196, Z -6.3333, A 0.000, B 0.000, C 0.000 }
gfCNCPoint4[23671] = {X 81.0151, Y 12.1868, Z -6.3333, A 0.000, B 0.000, C 0.000 }
gfCNCPoint4[23672] = {X 81.0160, Y 12.0923, Z -6.3333, A 0.000, B 0.000, C 0.000 }
gfCNCPoint4[23673] = {X 81.0187, Y 11.9978, Z -6.3333, A 0.000, B 0.000, C 0.000 }
gfCNCPoint4[23674] = {X 81.1325, Y 11.1229, Z -6.3333, A 0.000, B 0.000, C 0.000 }
gfCNCPoint4[23675] = {X 81.4018, Y 10.2828, Z -6.3333, A 0.000, B 0.000, C 0.000 }
gfCNCPoint4[23676] = {X 81.8181, Y 9.5049, Z -6.3333, A 0.000, B 0.000, C 0.000 }
gfCNCPoint4[23677] = {X 82.2191, Y 9.7687, Z -6.3333, A 0.000, B 0.000, C 0.000 }
gfCNCPoint4[23678] = {X 82.7659, Y 9.0935, Z -6.3333, A 0.000, B 0.000, C 0.000 }
gfCNCPoint4[23679] = {X 83.4348, Y 8.5389, Z -6.3333, A 0.000, B 0.000, C 0.000 }
gfCNCPoint4[23680] = {X 84.1996, Y 8.1266, Z -6.3333, A 0.000, B 0.000, C 0.000 }
gfCNCPoint4[23681] = {X 85.0305, Y 7.8726, Z -6.3333, A 0.000, B 0.000, C 0.000 }
gfCNCPoint4[23682] = {X 85.8951, Y 7.7868, Z -6.3333, A 0.000, B 0.000, C 0.000 }
gfCNCPoint4[23683] = {X 94.0497, Y 7.7868, Z -6.3333, A 0.000, B 0.000, C 0.000 }
gfCNCPoint4[23684] = {X 95.0288, Y 7.8971, Z -6.3333, A 0.000, B 0.000, C 0.000 }
gfCNCPoint4[23685] = {X 95.9588, Y 8.2226, Z -6.3333, A 0.000, B 0.000, C 0.000 }
gfCNCPoint4[23686] = {X 96.7930, Y 8.7468, Z -6.3333, A 0.000, B 0.000, C 0.000 }
gfCNCPoint4[23687] = {X 97.4897, Y 9.4435, Z -6.3333, A 0.000, B 0.000, C 0.000 }
gfCNCPoint4[23688] = {X 98.0139, Y 10.2777, Z -6.3333, A 0.000, B 0.000, C 0.000 }
gfCNCPoint4[23689] = {X 98.3394, Y 11.2077, Z -6.3333, A 0.000, B 0.000, C 0.000 }
gfCNCPoint4[23690] = {X 98.4497, Y 12.1868, Z -6.3333, A 0.000, B 0.000, C 0.000 }
gfCNCPoint4[23691] = {X 98.4494, Y 13.0233, Z -6.3333, A 0.000, B 0.000, C 0.000 }
gfCNCPoint4[23692] = {X 98.3724, Y 13.7989, Z -6.3333, A 0.000, B 0.000, C 0.000 }
gfCNCPoint4[23693] = {X 98.1598, Y 14.5487, Z -6.3333, A 0.000, B 0.000, C 0.000 }
gfCNCPoint4[23694] = {X 97.8182, Y 15.2493, Z -6.3333, A 0.000, B 0.000, C 0.000 }
gfCNCPoint4[23695] = {X 98.3686, Y 16.6194, Z -6.3333, A 0.000, B 0.000, C 0.000 }
gfCNCPoint4[23696] = {X 101.8746, Y 25.3103, Z -6.3333, A 0.000, B 0.000, C 0.000 }
gfCNCPoint4[23697] = {X 104.3483, Y 19.1464, Z -6.3333, A 0.000, B 0.000, C 0.000 }
gfCNCPoint4[23698] = {X 105.9236, Y 15.2221, Z -6.3333, A 0.000, B 0.000, C 0.000 }
gfCNCPoint4[23699] = {X 105.5854, Y 14.5149, Z -6.3333, A 0.000, B 0.000, C 0.000 }
gfCNCPoint4[23700] = {X 105.3781, Y 13.7588, Z -6.3333, A 0.000, B 0.000, C 0.000 }
gfCNCPoint4[23701] = {X 105.3083, Y 12.9780, Z -6.3333, A 0.000, B 0.000, C 0.000 }
gfCNCPoint4[23702] = {X 105.3083, Y 12.1868, Z -6.3333, A 0.000, B 0.000, C 0.000 }
gfCNCPoint4[23703] = {X 105.4186, Y 11.2077, Z -6.3333, A 0.000, B 0.000, C 0.000 }
gfCNCPoint4[23704] = {X 105.7440, Y 10.2777, Z -6.3333, A 0.000, B 0.000, C 0.000 }
gfCNCPoint4[23705] = {X 106.2682, Y 9.4435, Z -6.3333, A 0.000, B 0.000, C 0.000 }
gfCNCPoint4[23706] = {X 106.9649, Y 8.7468, Z -6.3333, A 0.000, B 0.000, C 0.000 }
gfCNCPoint4[23707] = {X 107.7992, Y 8.2226, Z -6.3333, A 0.000, B 0.000, C 0.000 }
gfCNCPoint4[23708] = {X 108.7292, Y 7.8971, Z -6.3333, A 0.000, B 0.000, C 0.000 }
gfCNCPoint4[23709] = {X 109.7083, Y 7.7868, Z -6.3333, A 0.000, B 0.000, C 0.000 }
gfCNCPoint4[23710] = {X 117.7916, Y 7.7868, Z -6.3333, A 0.000, B 0.000, C 0.000 }
gfCNCPoint4[23711] = {X 118.7707, Y 7.8971, Z -6.3333, A 0.000, B 0.000, C 0.000 }
gfCNCPoint4[23712] = {X 119.7007, Y 8.2226, Z -6.3333, A 0.000, B 0.000, C 0.000 }
gfCNCPoint4[23713] = {X 120.5349, Y 8.7468, Z -6.3333, A 0.000, B 0.000, C 0.000 }
gfCNCPoint4[23714] = {X 121.2316, Y 9.4435, Z -6.3333, A 0.000, B 0.000, C 0.000 }
gfCNCPoint4[23715] = {X 121.7558, Y 10.2777, Z -6.3333, A 0.000, B 0.000, C 0.000 }
gfCNCPoint4[23716] = {X 122.0813, Y 11.2077, Z -6.3333, A 0.000, B 0.000, C 0.000 }
gfCNCPoint4[23717] = {X 122.1916, Y 12.1868, Z -6.3333, A 0.000, B 0.000, C 0.000 }
gfCNCPoint4[23718] = {X 122.1913, Y 13.0233, Z -6.3333, A 0.000, B 0.000, C 0.000 }
gfCNCPoint4[23719] = {X 122.0831, Y 13.9490, Z -6.3333, A 0.000, B 0.000, C 0.000 }
gfCNCPoint4[23720] = {X 121.7823, Y 14.8311, Z -6.3333, A 0.000, B 0.000, C 0.000 }
gfCNCPoint4[23721] = {X 121.3025, Y 15.6301, Z -6.3333, A 0.000, B 0.000, C 0.000 }
gfCNCPoint4[23722] = {X 120.6651, Y 16.3101, Z -6.3333, A 0.000, B 0.000, C 0.000 }
gfCNCPoint4[23723] = {X 120.6647, Y 40.8767, Z -6.3333, A 0.000, B 0.000, C 0.000 }
gfCNCPoint4[23724] = {X 120.6784, Y 40.8882, Z -6.3333, A 0.000, B 0.000, C 0.000 }
gfCNCPoint4[23725] = {X 121.3172, Y 41.5763, Z -6.3333, A 0.000, B 0.000, C 0.000 }
gfCNCPoint4[23726] = {X 121.7955, Y 42.3843, Z -6.3333, A 0.000, B 0.000, C 0.000 }
gfCNCPoint4[23727] = {X 122.0914, Y 43.2753, Z -6.3333, A 0.000, B 0.000, C 0.000 }
gfCNCPoint4[23728] = {X 122.1916, Y 44.2089, Z -6.3333, A 0.000, B 0.000, C 0.000 }
gfCNCPoint4[23729] = {X 122.1916, Y 45.0000, Z -6.3333, A 0.000, B 0.000, C 0.000 }
gfCNCPoint4[23730] = {X 122.0813, Y 45.9791, Z -6.3333, A 0.000, B 0.000, C 0.000 }
gfCNCPoint4[23731] = {X 121.7558, Y 46.9091, Z -6.3333, A 0.000, B 0.000, C 0.000 }
gfCNCPoint4[23732] = {X 121.2316, Y 47.7434, Z -6.3333, A 0.000, B 0.000, C 0.000 }
gfCNCPoint4[23733] = {X 120.5349, Y 48.4401, Z -6.3333, A 0.000, B 0.000, C 0.000 }
gfCNCPoint4[23734] = {X 119.7007, Y 48.9643, Z -6.3333, A 0.000, B 0.000, C 0.000 }
gfCNCPoint4[23735] = {X 118.7707, Y 49.2897, Z -6.3333, A 0.000, B 0.000, C 0.000 }
gfCNCPoint4[23736] = {X 117.7916, Y 49.4000, Z -6.3333, A 0.000, B 0.000, C 0.000 }
gfCNCPoint4[23737] = {X 111.9185, Y 49.4000, Z -6.3333, A 0.000, B 0.000, C 0.000 }
gfCNCPoint4[23738] = {X 110.9394, Y 49.2897, Z -6.3333, A 0.000, B 0.000, C 0.000 }
gfCNCPoint4[23739] = {X 110.0094, Y 48.9643, Z -6.3333, A 0.000, B 0.000, C 0.000 }
gfCNCPoint4[23740] = {X 109.1751, Y 48.4400, Z -6.3333, A 0.000, B 0.000, C 0.000 }
gfCNCPoint4[23741] = {X 108.4784, Y 47.7433, Z -6.3333, A 0.000, B 0.000, C 0.000 }
gfCNCPoint4[23742] = {X 107.9542, Y 46.9091, Z -6.3333, A 0.000, B 0.000, C 0.000 }
gfCNCPoint4[23743] = {X 107.6288, Y 45.9791, Z -6.3333, A 0.000, B 0.000, C 0.000 }
gfCNCPoint4[23744] = {X 107.5185, Y 45.0000, Z -6.3333, A 0.000, B 0.000, C 0.000 }
gfCNCPoint4[23745] = {X 107.5185, Y 44.1789, Z -6.3333, A 0.000, B 0.000, C 0.000 }
gfCNCPoint4[23746] = {X 107.5547, Y 43.6261, Z -6.3333, A 0.000, B 0.000, C 0.000 }
gfCNCPoint4[23747] = {X 107.6627, Y 43.0828, Z -6.3333, A 0.000, B 0.000, C 0.000 }
gfCNCPoint4[23748] = {X 106.1856, Y 46.6923, Z -6.3333, A 0.000, B 0.000, C 0.000 }
gfCNCPoint4[23749] = {X 105.8087, Y 47.4049, Z -6.3333, A 0.000, B 0.000, C 0.000 }
gfCNCPoint4[23750] = {X 105.3081, Y 48.0367, Z -6.3333, A 0.000, B 0.000, C 0.000 }
gfCNCPoint4[23751] = {X 104.7006, Y 48.5667, Z -6.3333, A 0.000, B 0.000, C 0.000 }
gfCNCPoint4[23752] = {X 104.0067, Y 48.9769, Z -6.3333, A 0.000, B 0.000, C 0.000 }
gfCNCPoint4[23753] = {X 103.0414, Y 49.3033, Z -6.3333, A 0.000, B 0.000, C 0.000 }
gfCNCPoint4[23754] = {X 102.0269, Y 49.3989, Z -6.3333, A 0.000, B 0.000, C 0.000 }
gfCNCPoint4[23755] = {X 101.0176, Y 49.2586, Z -6.3333, A 0.000, B 0.000, C 0.000 }
gfCNCPoint4[23756] = {X 100.0676, Y 48.8899, Z -6.3333, A 0.000, B 0.000, C 0.000 }
gfCNCPoint4[23757] = {X 99.2280, Y 48.3125, Z -6.3333, A 0.000, B 0.000, C 0.000 }
gfCNCPoint4[23758] = {X 98.5436, Y 47.5575, Z -6.3333, A 0.000, B 0.000, C 0.000 }
gfCNCPoint4[23759] = {X 98.0514, Y 46.6653, Z -6.3333, A 0.000, B 0.000, C 0.000 }
gfCNCPoint4[23760] = {X 96.5886, Y 43.0879, Z -6.3333, A 0.000, B 0.000, C 0.000 }
gfCNCPoint4[23761] = {X 96.6991, Y 43.6436, Z -6.3333, A 0.000, B 0.000, C 0.000 }
gfCNCPoint4[23762] = {X 96.7385, Y 44.2089, Z -6.3333, A 0.000, B 0.000, C 0.000 }
gfCNCPoint4[23763] = {X 96.7383, Y 45.0423, Z -6.3333, A 0.000, B 0.000, C 0.000 }
gfCNCPoint4[23764] = {X 96.6200, Y 46.0144, Z -6.3333, A 0.000, B 0.000, C 0.000 }
gfCNCPoint4[23765] = {X 96.2896, Y 46.9363, Z -6.3333, A 0.000, B 0.000, C 0.000 }
gfCNCPoint4[23766] = {X 95.7635, Y 47.7622, Z -6.3333, A 0.000, B 0.000, C 0.000 }
gfCNCPoint4[23767] = {X 95.0677, Y 48.4513, Z -6.3333, A 0.000, B 0.000, C 0.000 }
gfCNCPoint4[23768] = {X 94.2367, Y 48.9695, Z -6.3333, A 0.000, B 0.000, C 0.000 }
gfCNCPoint4[23769] = {X 93.3117, Y 49.2910, Z -6.3333, A 0.000, B 0.000, C 0.000 }
gfCNCPoint4[23770] = {X 92.3385, Y 49.4000, Z -6.3333, A 0.000, B 0.000, C 0.000 }
gfCNCPoint4[23771] = {X 85.8951, Y 49.4000, Z -6.3333, A 0.000, B 0.000, C 0.000 }
gfCNCPoint4[23772] = {X 84.9160, Y 49.2897, Z -6.3333, A 0.000, B 0.000, C 0.000 }
gfCNCPoint4[23773] = {X 83.9860, Y 48.9643, Z -6.3333, A 0.000, B 0.000, C 0.000 }
gfCNCPoint4[23774] = {X 83.1517, Y 48.4400, Z -6.3333, A 0.000, B 0.000, C 0.000 }
gfCNCPoint4[23775] = {X 82.4550, Y 47.7433, Z -6.3333, A 0.000, B 0.000, C 0.000 }
gfCNCPoint4[23776] = {X 81.9308, Y 46.9091, Z -6.3333, A 0.000, B 0.000, C 0.000 }
gfCNCPoint4[23777] = {X 81.6054, Y 45.9791, Z -6.3333, A 0.000, B 0.000, C 0.000 }
gfCNCPoint4[23778] = {X 81.4951, Y 45.0000, Z -6.3333, A 0.000, B 0.000, C 0.000 }
gfCNCPoint4[23779] = {X 81.4951, Y 44.2067, Z -6.3333, A 0.000, B 0.000, C 0.000 }
gfCNCPoint4[23780] = {X 81.5999, Y 43.2694, Z -6.3333, A 0.000, B 0.000, C 0.000 }
gfCNCPoint4[23781] = {X 81.8996, Y 42.3750, Z -6.3333, A 0.000, B 0.000, C 0.000 }
gfCNCPoint4[23782] = {X 82.3809, Y 41.5639, Z -6.3333, A 0.000, B 0.000, C 0.000 }
gfCNCPoint4[23783] = {X 83.0222, Y 40.8722, Z -6.3333, A 0.000, B 0.000, C 0.000 }
gfCNCPoint4[23784] = {X 83.0219, Y 16.3104, Z -6.3333, A 0.000, B 0.000, C 0.000 }
gfCNCPoint4[23785] = {X 82.3776, Y 15.6213, Z -6.3333, A 0.000, B 0.000, C 0.000 }
gfCNCPoint4[23786] = {X 81.8949, Y 14.8108, Z -6.3333, A 0.000, B 0.000, C 0.000 }
gfCNCPoint4[23787] = {X 81.5962, Y 13.9159, Z -6.3333, A 0.000, B 0.000, C 0.000 }
gfCNCPoint4[23788] = {X 81.4951, Y 12.9780, Z -6.3333, A 0.000, B 0.000, C 0.000 }
gfCNCPoint4[23789] = {X 81.4951, Y 12.1868, Z -6.3333, A 0.000, B 0.000, C 0.000 }
gfCNCPoint4[23790] = {X 81.5776, Y 11.3388, Z -6.3333, A 0.000, B 0.000, C 0.000 }
gfCNCPoint4[23791] = {X 81.8220, Y 10.5225, Z -6.3333, A 0.000, B 0.000, C 0.000 }
gfCNCPoint4[23792] = {X 82.2191, Y 9.7687, Z -6.3333, A 0.000, B 0.000, C 0.000 }
gfCNCPoint4[23793] = {X 81.8181, Y 9.5049, Z -6.3333, A 0.000, B 0.000, C 0.000 }
gfCNCPoint4[23794] = {X 68.9232, Y 9.5049, Z -6.3333, A 0.000, B 0.000, C 0.000 }
gfCNCPoint4[23795] = {X 69.1905, Y 10.7208, Z -6.3333, A 0.000, B 0.000, C 0.000 }
gfCNCPoint4[23796] = {X 69.2995, Y 11.9609, Z -6.3333, A 0.000, B 0.000, C 0.000 }
gfCNCPoint4[23797] = {X 69.3015, Y 12.0739, Z -6.3333, A 0.000, B 0.000, C 0.000 }
gfCNCPoint4[23798] = {X 69.3021, Y 12.1868, Z -6.3333, A 0.000, B 0.000, C 0.000 }
gfCNCPoint4[23799] = {X 69.3017, Y 13.0686, Z -6.3333, A 0.000, B 0.000, C 0.000 }
gfCNCPoint4[23800] = {X 69.2128, Y 14.2901, Z -6.3333, A 0.000, B 0.000, C 0.000 }
gfCNCPoint4[23801] = {X 68.9704, Y 15.4905, Z -6.3333, A 0.000, B 0.000, C 0.000 }
gfCNCPoint4[23802] = {X 73.2459, Y 26.9277, Z -6.3333, A 0.000, B 0.000, C 0.000 }
gfCNCPoint4[23803] = {X 77.7420, Y 25.2469, Z -6.3333, A 0.000, B 0.000, C 0.000 }
gfCNCPoint4[23804] = {X 77.7419, Y 18.1961, Z -6.3333, A 0.000, B 0.000, C 0.000 }
gfCNCPoint4[23805] = {X 77.0777, Y 16.9727, Z -6.3333, A 0.000, B 0.000, C 0.000 }
gfCNCPoint4[23806] = {X 76.5959, Y 15.6666, Z -6.3333, A 0.000, B 0.000, C 0.000 }
gfCNCPoint4[23807] = {X 76.3064, Y 14.3049, Z -6.3333, A 0.000, B 0.000, C 0.000 }
gfCNCPoint4[23808] = {X 74.0412, Y 14.3049, Z -6.3333, A 0.000, B 0.000, C 0.000 }
gfCNCPoint4[23809] = {X 73.9993, Y 14.7002, Z -6.3333, A 0.000, B 0.000, C 0.000 }
gfCNCPoint4[23810] = {X 73.9466, Y 15.0942, Z -6.3333, A 0.000, B 0.000, C 0.000 }
gfCNCPoint4[23811] = {X 77.7420, Y 25.2469, Z -6.3333, A 0.000, B 0.000, C 0.000 }
gfCNCPoint4[23812] = {X 75.4940, Y 26.0873, Z -6.3333, A 0.000, B 0.000, C 0.000 }
gfCNCPoint4[23813] = {X 78.9563, Y 35.3492, Z -6.3333, A 0.000, B 0.000, C 0.000 }
gfCNCPoint4[23814] = {X 79.5721, Y 35.9626, Z -6.3333, A 0.000, B 0.000, C 0.000 }
gfCNCPoint4[23815] = {X 80.1421, Y 36.6187, Z -6.3333, A 0.000, B 0.000, C 0.000 }
gfCNCPoint4[23816] = {X 80.1419, Y 17.4389, Z -6.3333, A 0.000, B 0.000, C 0.000 }
gfCNCPoint4[23817] = {X 79.4939, Y 16.4455, Z -6.3333, A 0.000, B 0.000, C 0.000 }
gfCNCPoint4[23818] = {X 79.0158, Y 15.3601, Z -6.3333, A 0.000, B 0.000, C 0.000 }
gfCNCPoint4[23819] = {X 78.7203, Y 14.2115, Z -6.3333, A 0.000, B 0.000, C 0.000 }
gfCNCPoint4[23820] = {X 78.6153, Y 13.0301, Z -6.3333, A 0.000, B 0.000, C 0.000 }
gfCNCPoint4[23821] = {X 78.6151, Y 12.1868, Z -6.3333, A 0.000, B 0.000, C 0.000 }
gfCNCPoint4[23822] = {X 78.6164, Y 12.0458, Z -6.3333, A 0.000, B 0.000, C 0.000 }
gfCNCPoint4[23823] = {X 78.6205, Y 11.9049, Z -6.3333, A 0.000, B 0.000, C 0.000 }
gfCNCPoint4[23824] = {X 71.6988, Y 11.9049, Z -6.3333, A 0.000, B 0.000, C 0.000 }
gfCNCPoint4[23825] = {X 71.7013, Y 12.0458, Z -6.3333, A 0.000, B 0.000, C 0.000 }
gfCNCPoint4[23826] = {X 71.7021, Y 12.1868, Z -6.3333, A 0.000, B 0.000, C 0.000 }
gfCNCPoint4[23827] = {X 71.7016, Y 13.0911, Z -6.3333, A 0.000, B 0.000, C 0.000 }
gfCNCPoint4[23828] = {X 71.6387, Y 14.2145, Z -6.3333, A 0.000, B 0.000, C 0.000 }
gfCNCPoint4[23829] = {X 71.4715, Y 15.3272, Z -6.3333, A 0.000, B 0.000, C 0.000 }
gfCNCPoint4[23830] = {X 75.4940, Y 26.0873, Z -6.3333, A 0.000, B 0.000, C 0.000 }
gfCNCPoint4[23831] = {X 73.2459, Y 26.9277, Z -6.3333, A 0.000, B 0.000, C 0.000 }
gfCNCPoint4[23832] = {X 76.9192, Y 36.7539, Z -6.3333, A 0.000, B 0.000, C 0.000 }
gfCNCPoint4[23833] = {X 77.6314, Y 37.4064, Z -6.3333, A 0.000, B 0.000, C 0.000 }
gfCNCPoint4[23834] = {X 78.2750, Y 38.1266, Z -6.3333, A 0.000, B 0.000, C 0.000 }
gfCNCPoint4[23835] = {X 79.0227, Y 39.1916, Z -6.3333, A 0.000, B 0.000, C 0.000 }
gfCNCPoint4[23836] = {X 79.6209, Y 40.3472, Z -6.3333, A 0.000, B 0.000, C 0.000 }
gfCNCPoint4[23837] = {X 80.0586, Y 41.5725, Z -6.3333, A 0.000, B 0.000, C 0.000 }
gfCNCPoint4[23838] = {X 80.3280, Y 42.8455, Z -6.3333, A 0.000, B 0.000, C 0.000 }
gfCNCPoint4[23839] = {X 80.4242, Y 44.1432, Z -6.3333, A 0.000, B 0.000, C 0.000 }
gfCNCPoint4[23840] = {X 80.4245, Y 45.0000, Z -6.3333, A 0.000, B 0.000, C 0.000 }
gfCNCPoint4[23841] = {X 80.3511, Y 46.1898, Z -6.3333, A 0.000, B 0.000, C 0.000 }
gfCNCPoint4[23842] = {X 80.1320, Y 47.3615, Z -6.3333, A 0.000, B 0.000, C 0.000 }
gfCNCPoint4[23843] = {X 79.7706, Y 48.4974, Z -6.3333, A 0.000, B 0.000, C 0.000 }
gfCNCPoint4[23844] = {X 79.2722, Y 49.5803, Z -6.3333, A 0.000, B 0.000, C 0.000 }
gfCNCPoint4[23845] = {X 78.4688, Y 50.8341, Z -6.3333, A 0.000, B 0.000, C 0.000 }
gfCNCPoint4[23846] = {X 77.4826, Y 51.9498, Z -6.3333, A 0.000, B 0.000, C 0.000 }
gfCNCPoint4[23847] = {X 76.3369, Y 52.9011, Z -6.3333, A 0.000, B 0.000, C 0.000 }
gfCNCPoint4[23848] = {X 75.0589, Y 53.6653, Z -6.3333, A 0.000, B 0.000, C 0.000 }
gfCNCPoint4[23849] = {X 73.6787, Y 54.2246, Z -6.3333, A 0.000, B 0.000, C 0.000 }
gfCNCPoint4[23850] = {X 72.2292, Y 54.5655, Z -6.3333, A 0.000, B 0.000, C 0.000 }
gfCNCPoint4[23851] = {X 70.7445, Y 54.6800, Z -6.3333, A 0.000, B 0.000, C 0.000 }
gfCNCPoint4[23852] = {X 64.1851, Y 54.6800, Z -6.3333, A 0.000, B 0.000, C 0.000 }
gfCNCPoint4[23853] = {X 62.7229, Y 54.5689, Z -6.3333, A 0.000, B 0.000, C 0.000 }
gfCNCPoint4[23854] = {X 61.2943, Y 54.2383, Z -6.3333, A 0.000, B 0.000, C 0.000 }
gfCNCPoint4[23855] = {X 59.9320, Y 53.6956, Z -6.3333, A 0.000, B 0.000, C 0.000 }
gfCNCPoint4[23856] = {X 58.6673, Y 52.9534, Z -6.3333, A 0.000, B 0.000, C 0.000 }
gfCNCPoint4[23857] = {X 57.5293, Y 52.0286, Z -6.3333, A 0.000, B 0.000, C 0.000 }
gfCNCPoint4[23858] = {X 56.6337, Y 51.0563, Z -6.3333, A 0.000, B 0.000, C 0.000 }
gfCNCPoint4[23859] = {X 55.8790, Y 49.9710, Z -6.3333, A 0.000, B 0.000, C 0.000 }
gfCNCPoint4[23860] = {X 55.1243, Y 51.0563, Z -6.3333, A 0.000, B 0.000, C 0.000 }
gfCNCPoint4[23861] = {X 54.2288, Y 52.0286, Z -6.3333, A 0.000, B 0.000, C 0.000 }
gfCNCPoint4[23862] = {X 53.0907, Y 52.9534, Z -6.3333, A 0.000, B 0.000, C 0.000 }
gfCNCPoint4[23863] = {X 51.8261, Y 53.6956, Z -6.3333, A 0.000, B 0.000, C 0.000 }
gfCNCPoint4[23864] = {X 50.4638, Y 54.2383, Z -6.3333, A 0.000, B 0.000, C 0.000 }
gfCNCPoint4[23865] = {X 49.0351, Y 54.5689, Z -6.3333, A 0.000, B 0.000, C 0.000 }
gfCNCPoint4[23866] = {X 47.5729, Y 54.6800, Z -6.3333, A 0.000, B 0.000, C 0.000 }
gfCNCPoint4[23867] = {X 40.6393, Y 54.6800, Z -6.3333, A 0.000, B 0.000, C 0.000 }
gfCNCPoint4[23868] = {X 39.2448, Y 54.5790, Z -6.3333, A 0.000, B 0.000, C 0.000 }
gfCNCPoint4[23869] = {X 37.8793, Y 54.2782, Z -6.3333, A 0.000, B 0.000, C 0.000 }
gfCNCPoint4[23870] = {X 36.5715, Y 53.7838, Z -6.3333, A 0.000, B 0.000, C 0.000 }
gfCNCPoint4[23871] = {X 35.3485, Y 53.1062, Z -6.3333, A 0.000, B 0.000, C 0.000 }
gfCNCPoint4[23872] = {X 33.9150, Y 54.1349, Z -6.3333, A 0.000, B 0.000, C 0.000 }
gfCNCPoint4[23873] = {X 32.3635, Y 54.9754, Z -6.3333, A 0.000, B 0.000, C 0.000 }
gfCNCPoint4[23874] = {X 30.7187, Y 55.6142, Z -6.3333, A 0.000, B 0.000, C 0.000 }
gfCNCPoint4[23875] = {X 29.0066, Y 56.0411, Z -6.3333, A 0.000, B 0.000, C 0.000 }
gfCNCPoint4[23876] = {X 27.2545, Y 56.2496, Z -6.3333, A 0.000, B 0.000, C 0.000 }
gfCNCPoint4[23877] = {X 24.9802, Y 57.2328, Z -6.3333, A 0.000, B 0.000, C 0.000 }
gfCNCPoint4[23878] = {X 22.6482, Y 58.0699, Z -6.3333, A 0.000, B 0.000, C 0.000 }
gfCNCPoint4[23879] = {X 20.0861, Y 58.7989, Z -6.3333, A 0.000, B 0.000, C 0.000 }
gfCNCPoint4[23880] = {X 17.4729, Y 59.3152, Z -6.3333, A 0.000, B 0.000, C 0.000 }
gfCNCPoint4[23881] = {X 14.8261, Y 59.6153, Z -6.3333, A 0.000, B 0.000, C 0.000 }
gfCNCPoint4[23882] = {X 12.1636, Y 59.6973, Z -6.3333, A 0.000, B 0.000, C 0.000 }
gfCNCPoint4[23883] = {X 9.5034, Y 59.5604, Z -6.3333, A 0.000, B 0.000, C 0.000 }
gfCNCPoint4[23884] = {X 9.5034, Y 90.4951, Z -6.3333, A 0.000, B 0.000, C 0.000 }
gfCNCPoint4[23885] = {X 114.8634, Y 90.4951, Z -6.3333, A 0.000, B 0.000, C 0.000 }
gfCNCPoint4[23886] = {X 115.7476, Y 89.2994, Z -6.3333, A 0.000, B 0.000, C 0.000 }
gfCNCPoint4[23887] = {X 116.7721, Y 88.2213, Z -6.3333, A 0.000, B 0.000, C 0.000 }
gfCNCPoint4[23888] = {X 117.9212, Y 87.2773, Z -6.3333, A 0.000, B 0.000, C 0.000 }
gfCNCPoint4[23889] = {X 119.1776, Y 86.4817, Z -6.3333, A 0.000, B 0.000, C 0.000 }
gfCNCPoint4[23890] = {X 120.5223, Y 85.8465, Z -6.3333, A 0.000, B 0.000, C 0.000 }
gfCNCPoint4[23891] = {X 121.9348, Y 85.3813, Z -6.3333, A 0.000, B 0.000, C 0.000 }
gfCNCPoint4[23892] = {X 123.3938, Y 85.0932, Z -6.3333, A 0.000, B 0.000, C 0.000 }
gfCNCPoint4[23893] = {X 123.5618, Y 84.9123, Z -6.3333, A 0.000, B 0.000, C 0.000 }
gfCNCPoint4[23894] = {X 123.7279, Y 84.7295, Z -6.3333, A 0.000, B 0.000, C 0.000 }
gfCNCPoint4[23895] = {X 147.2181, Y 58.9341, Z -6.3333, A 0.000, B 0.000, C 0.000 }
gfCNCPoint4[23896] = {X 147.2180, Y 58.0000, Z -6.3333, A 0.000, B 0.000, C 0.000 }
gfCNCPoint4[23897] = {X 147.2987, Y 56.6058, Z -6.3333, A 0.000, B 0.000, C 0.000 }
gfCNCPoint4[23898] = {X 147.5398, Y 55.2303, Z -6.3333, A 0.000, B 0.000, C 0.000 }
gfCNCPoint4[23899] = {X 148.0022, Y 53.7185, Z -6.3333, A 0.000, B 0.000, C 0.000 }
gfCNCPoint4[23900] = {X 148.6580, Y 52.2800, Z -6.3333, A 0.000, B 0.000, C 0.000 }
gfCNCPoint4[23901] = {X 143.0396, Y 52.2800, Z -6.3333, A 0.000, B 0.000, C 0.000 }
gfCNCPoint4[23902] = {X 141.7807, Y 52.1703, Z -6.3333, A 0.000, B 0.000, C 0.000 }
gfCNCPoint4[23903] = {X 140.5597, Y 51.8446, Z -6.3333, A 0.000, B 0.000, C 0.000 }
gfCNCPoint4[23904] = {X 139.4134, Y 51.3126, Z -6.3333, A 0.000, B 0.000, C 0.000 }
gfCNCPoint4[23905] = {X 138.3764, Y 50.5904, Z -6.3333, A 0.000, B 0.000, C 0.000 }
gfCNCPoint4[23906] = {X 137.4799, Y 49.6998, Z -6.3333, A 0.000, B 0.000, C 0.000 }
gfCNCPoint4[23907] = {X 136.7509, Y 48.6675, Z -6.3333, A 0.000, B 0.000, C 0.000 }
gfCNCPoint4[23908] = {X 136.2114, Y 47.5248, Z -6.3333, A 0.000, B 0.000, C 0.000 }
gfCNCPoint4[23909] = {X 135.8777, Y 46.3059, Z -6.3333, A 0.000, B 0.000, C 0.000 }
gfCNCPoint4[23910] = {X 135.7598, Y 45.0477, Z -6.3333, A 0.000, B 0.000, C 0.000 }
gfCNCPoint4[23911] = {X 135.7601, Y 44.1247, Z -6.3333, A 0.000, B 0.000, C 0.000 }
gfCNCPoint4[23912] = {X 135.8408, Y 43.1249, Z -6.3333, A 0.000, B 0.000, C 0.000 }
gfCNCPoint4[23913] = {X 136.0581, Y 42.1457, Z -6.3333, A 0.000, B 0.000, C 0.000 }
gfCNCPoint4[23914] = {X 138.3597, Y 42.8258, Z -6.3333, A 0.000, B 0.000, C 0.000 }
gfCNCPoint4[23915] = {X 138.6721, Y 42.0319, Z -6.3333, A 0.000, B 0.000, C 0.000 }
gfCNCPoint4[23916] = {X 139.1179, Y 41.3046, Z -6.3333, A 0.000, B 0.000, C 0.000 }
gfCNCPoint4[23917] = {X 139.6836, Y 40.6660, Z -6.3333, A 0.000, B 0.000, C 0.000 }
gfCNCPoint4[23918] = {X 139.6836, Y 20.4379, Z -6.3333, A 0.000, B 0.000, C 0.000 }
gfCNCPoint4[23919] = {X 137.7098, Y 20.4376, Z -6.3333, A 0.000, B 0.000, C 0.000 }
gfCNCPoint4[23920] = {X 136.9997, Y 21.1825, Z -6.3333, A 0.000, B 0.000, C 0.000 }
gfCNCPoint4[23921] = {X 136.1491, Y 21.7619, Z -6.3333, A 0.000, B 0.000, C 0.000 }
gfCNCPoint4[23922] = {X 135.4282, Y 22.0767, Z -6.3333, A 0.000, B 0.000, C 0.000 }
gfCNCPoint4[23923] = {X 134.6660, Y 22.2715, Z -6.3333, A 0.000, B 0.000, C 0.000 }
gfCNCPoint4[23924] = {X 133.8824, Y 22.3414, Z -6.3333, A 0.000, B 0.000, C 0.000 }
gfCNCPoint4[23925] = {X 133.2006, Y 22.3415, Z -6.3333, A 0.000, B 0.000, C 0.000 }
gfCNCPoint4[23926] = {X 132.2486, Y 22.2478, Z -6.3333, A 0.000, B 0.000, C 0.000 }
gfCNCPoint4[23927] = {X 131.3331, Y 21.9701, Z -6.3333, A 0.000, B 0.000, C 0.000 }
gfCNCPoint4[23928] = {X 130.4895, Y 21.5191, Z -6.3333, A 0.000, B 0.000, C 0.000 }
gfCNCPoint4[23929] = {X 129.7500, Y 20.9122, Z -6.3333, A 0.000, B 0.000, C 0.000 }
gfCNCPoint4[23930] = {X 129.1431, Y 20.1727, Z -6.3333, A 0.000, B 0.000, C 0.000 }
gfCNCPoint4[23931] = {X 128.6921, Y 19.3290, Z -6.3333, A 0.000, B 0.000, C 0.000 }
gfCNCPoint4[23932] = {X 128.4144, Y 18.4136, Z -6.3333, A 0.000, B 0.000, C 0.000 }
gfCNCPoint4[23933] = {X 128.3206, Y 17.4615, Z -6.3333, A 0.000, B 0.000, C 0.000 }
gfCNCPoint4[23934] = {X 128.3206, Y 10.4835, Z -6.3333, A 0.000, B 0.000, C 0.000 }
gfCNCPoint4[23935] = {X 128.3317, Y 10.1548, Z -6.3333, A 0.000, B 0.000, C 0.000 }
gfCNCPoint4[23936] = {X 128.3649, Y 9.8275, Z -6.3333, A 0.000, B 0.000, C 0.000 }
gfCNCPoint4[23937] = {X 128.6079, Y 8.8340, Z -6.3333, A 0.000, B 0.000, C 0.000 }
gfCNCPoint4[23938] = {X 129.0525, Y 7.9130, Z -6.3333, A 0.000, B 0.000, C 0.000 }
gfCNCPoint4[23939] = {X 129.6794, Y 7.1049, Z -6.3333, A 0.000, B 0.000, C 0.000 }
gfCNCPoint4[23940] = {X 130.0257, Y 7.4372, Z -6.3333, A 0.000, B 0.000, C 0.000 }
gfCNCPoint4[23941] = {X 130.6997, Y 6.8634, Z -6.3333, A 0.000, B 0.000, C 0.000 }
gfCNCPoint4[23942] = {X 131.4749, Y 6.4361, Z -6.3333, A 0.000, B 0.000, C 0.000 }
gfCNCPoint4[23943] = {X 132.3200, Y 6.1726, Z -6.3333, A 0.000, B 0.000, C 0.000 }
gfCNCPoint4[23944] = {X 133.2007, Y 6.0835, Z -6.3333, A 0.000, B 0.000, C 0.000 }
gfCNCPoint4[23945] = {X 133.8874, Y 6.0837, Z -6.3333, A 0.000, B 0.000, C 0.000 }
gfCNCPoint4[23946] = {X 134.7187, Y 6.1717, Z -6.3333, A 0.000, B 0.000, C 0.000 }
gfCNCPoint4[23947] = {X 135.5183, Y 6.4152, Z -6.3333, A 0.000, B 0.000, C 0.000 }
gfCNCPoint4[23948] = {X 136.2575, Y 6.8056, Z -6.3333, A 0.000, B 0.000, C 0.000 }
gfCNCPoint4[23949] = {X 136.9094, Y 7.3287, Z -6.3333, A 0.000, B 0.000, C 0.000 }
gfCNCPoint4[23950] = {X 137.4507, Y 7.9657, Z -6.3333, A 0.000, B 0.000, C 0.000 }
gfCNCPoint4[23951] = {X 155.0720, Y 7.9657, Z -6.3333, A 0.000, B 0.000, C 0.000 }
gfCNCPoint4[23952] = {X 155.6198, Y 7.3224, Z -6.3333, A 0.000, B 0.000, C 0.000 }
gfCNCPoint4[23953] = {X 156.2804, Y 6.7957, Z -6.3333, A 0.000, B 0.000, C 0.000 }
gfCNCPoint4[23954] = {X 157.0295, Y 6.4050, Z -6.3333, A 0.000, B 0.000, C 0.000 }
gfCNCPoint4[23955] = {X 157.8395, Y 6.1646, Z -6.3333, A 0.000, B 0.000, C 0.000 }
gfCNCPoint4[23956] = {X 158.6805, Y 6.0835, Z -6.3333, A 0.000, B 0.000, C 0.000 }
gfCNCPoint4[23957] = {X 159.3791, Y 6.0839, Z -6.3333, A 0.000, B 0.000, C 0.000 }
gfCNCPoint4[23958] = {X 160.3488, Y 6.2050, Z -6.3333, A 0.000, B 0.000, C 0.000 }
gfCNCPoint4[23959] = {X 161.2678, Y 6.5371, Z -6.3333, A 0.000, B 0.000, C 0.000 }
gfCNCPoint4[23960] = {X 162.0908, Y 7.0639, Z -6.3333, A 0.000, B 0.000, C 0.000 }
gfCNCPoint4[23961] = {X 162.7773, Y 7.7593, Z -6.3333, A 0.000, B 0.000, C 0.000 }
gfCNCPoint4[23962] = {X 163.2934, Y 8.5891, Z -6.3333, A 0.000, B 0.000, C 0.000 }
gfCNCPoint4[23963] = {X 163.6136, Y 9.5124, Z -6.3333, A 0.000, B 0.000, C 0.000 }
gfCNCPoint4[23964] = {X 163.7221, Y 10.4835, Z -6.3333, A 0.000, B 0.000, C 0.000 }
gfCNCPoint4[23965] = {X 163.7221, Y 17.4615, Z -6.3333, A 0.000, B 0.000, C 0.000 }
gfCNCPoint4[23966] = {X 163.6118, Y 18.4406, Z -6.3333, A 0.000, B 0.000, C 0.000 }
gfCNCPoint4[23967] = {X 163.2863, Y 19.3706, Z -6.3333, A 0.000, B 0.000, C 0.000 }
gfCNCPoint4[23968] = {X 162.7621, Y 20.2049, Z -6.3333, A 0.000, B 0.000, C 0.000 }
gfCNCPoint4[23969] = {X 162.0654, Y 20.9016, Z -6.3333, A 0.000, B 0.000, C 0.000 }
gfCNCPoint4[23970] = {X 161.2312, Y 21.4258, Z -6.3333, A 0.000, B 0.000, C 0.000 }
gfCNCPoint4[23971] = {X 160.3012, Y 21.7512, Z -6.3333, A 0.000, B 0.000, C 0.000 }
gfCNCPoint4[23972] = {X 159.3221, Y 21.8615, Z -6.3333, A 0.000, B 0.000, C 0.000 }
gfCNCPoint4[23973] = {X 158.6790, Y 21.8615, Z -6.3333, A 0.000, B 0.000, C 0.000 }
gfCNCPoint4[23974] = {X 157.8335, Y 21.7770, Z -6.3333, A 0.000, B 0.000, C 0.000 }
gfCNCPoint4[23975] = {X 157.0197, Y 21.5326, Z -6.3333, A 0.000, B 0.000, C 0.000 }
gfCNCPoint4[23976] = {X 156.2676, Y 21.1374, Z -6.3333, A 0.000, B 0.000, C 0.000 }
gfCNCPoint4[23977] = {X 155.6046, Y 20.6059, Z -6.3333, A 0.000, B 0.000, C 0.000 }
gfCNCPoint4[23978] = {X 155.0553, Y 19.9576, Z -6.3333, A 0.000, B 0.000, C 0.000 }
gfCNCPoint4[23979] = {X 152.3569, Y 19.9586, Z -6.3333, A 0.000, B 0.000, C 0.000 }
gfCNCPoint4[23980] = {X 152.3558, Y 40.8428, Z -6.3333, A 0.000, B 0.000, C 0.000 }
gfCNCPoint4[23981] = {X 152.8072, Y 41.3296, Z -6.3333, A 0.000, B 0.000, C 0.000 }
gfCNCPoint4[23982] = {X 152.9007, Y 41.4409, Z -6.3333, A 0.000, B 0.000, C 0.000 }
gfCNCPoint4[23983] = {X 153.4351, Y 42.2812, Z -6.3333, A 0.000, B 0.000, C 0.000 }
gfCNCPoint4[23984] = {X 153.7682, Y 43.2197, Z -6.3333, A 0.000, B 0.000, C 0.000 }
gfCNCPoint4[23985] = {X 153.8831, Y 44.2089, Z -6.3333, A 0.000, B 0.000, C 0.000 }
gfCNCPoint4[23986] = {X 153.8829, Y 45.0423, Z -6.3333, A 0.000, B 0.000, C 0.000 }
gfCNCPoint4[23987] = {X 153.7646, Y 46.0144, Z -6.3333, A 0.000, B 0.000, C 0.000 }
gfCNCPoint4[23988] = {X 153.4342, Y 46.9363, Z -6.3333, A 0.000, B 0.000, C 0.000 }
gfCNCPoint4[23989] = {X 152.9080, Y 47.7622, Z -6.3333, A 0.000, B 0.000, C 0.000 }
gfCNCPoint4[23990] = {X 152.2123, Y 48.4513, Z -6.3333, A 0.000, B 0.000, C 0.000 }
gfCNCPoint4[23991] = {X 151.3813, Y 48.9695, Z -6.3333, A 0.000, B 0.000, C 0.000 }
gfCNCPoint4[23992] = {X 150.4563, Y 49.2910, Z -6.3333, A 0.000, B 0.000, C 0.000 }
gfCNCPoint4[23993] = {X 149.4831, Y 49.4000, Z -6.3333, A 0.000, B 0.000, C 0.000 }
gfCNCPoint4[23994] = {X 143.0396, Y 49.4000, Z -6.3333, A 0.000, B 0.000, C 0.000 }
gfCNCPoint4[23995] = {X 142.0605, Y 49.2897, Z -6.3333, A 0.000, B 0.000, C 0.000 }
gfCNCPoint4[23996] = {X 141.1305, Y 48.9643, Z -6.3333, A 0.000, B 0.000, C 0.000 }
gfCNCPoint4[23997] = {X 140.2963, Y 48.4400, Z -6.3333, A 0.000, B 0.000, C 0.000 }
gfCNCPoint4[23998] = {X 139.5996, Y 47.7433, Z -6.3333, A 0.000, B 0.000, C 0.000 }
gfCNCPoint4[23999] = {X 139.0754, Y 46.9091, Z -6.3333, A 0.000, B 0.000, C 0.000 }
